# B&R Automation Studio project vibratorControlWithCurrentController (part 13)

#### machine.st - Init, cyclic, exit code
```iecst
PROGRAM _INIT
	cm.setup.name := 'machine';
	cm.setup.parent.name := 'main';

	this.CfgSetIPAddr_0.Option  := cfgOPTION_NON_VOLATILE;
	//this.hmi.setNtpClient := TRUE;

	ST_name(0,ADR(this.configName),0);
	brdkStrCat(ADR(this.configName),ADR(':this.hmi.config'));

	this.hmi.config.dhcpEnabled := TRUE;

	this.TON_updateIp.PT := T#30s;

//	this.forceOutputsFB[0].dpName  := '%QX.IF6.ST6.DigitalOutput01'; //main:this.hw.do_stopButtonIndicator
//	this.forceOutputsFB[1].dpName  := '%QX.IF6.ST6.DigitalOutput02'; //main:this.hw.do_startButtonIndicator
	this.forceOutputsFB[2].dpName  := '%QX.IF6.ST2.DigitalOutput02'; //main:this.hw.do_alarmBeacon
	//this.forceOutputsFB[3].dpName  := '%QX.IF6.ST13.DigitalOutput01'; //feeder:this.hw.do_beltForwards
	//this.forceOutputsFB[4].dpName  := '%QX.IF6.ST13.DigitalOutput02'; //feeder:this.hw.do_beltBackwards
	this.forceOutputsFB[5].dpName  := '%QX.IF6.ST2.DigitalOutput01'; //feeder:this.hw.do_levelSensorInBowlLow
	this.forceOutputsFB[6].dpName  := '%QX.IF6.ST2.DigitalOutput03'; //feeder:this.hw.do_levelSensorInBowlMedium
	this.forceOutputsFB[7].dpName  := '%QX.IF6.ST2.DigitalOutput05'; //feeder:this.hw.do_levelSensorInBowlHigh

	this.forceOutputsFB[8].dpName  := '%QX.IF6.ST7.DigitalOutput01'; //upperFlap:this.hw.do_open
	this.forceOutputsFB[9].dpName  := '%QX.IF6.ST7.DigitalOutput03'; //middleFlap:this.hw.do_open
	this.forceOutputsFB[10].dpName := '%QX.IF6.ST8.DigitalOutput01'; //bottomFlap:this.hw.do_open
	this.forceOutputsFB[11].dpName := '%QX.IF6.ST8.DigitalOutput03'; //bottomFlap:this.hw.do_neighbourOpen
	this.forceOutputsFB[12].dpName := '%QX.IF6.ST7.DigitalOutput04'; //cassette:this.hw.do_dosing
	this.forceOutputsFB[13].dpName := '%QX.IF6.ST8.DigitalOutput05'; //cassette:this.hw.do_cassetteRelease
	this.forceOutputsFB[14].dpName := '%QX.IF6.ST7.DigitalOutput07'; //cassette:this.hw.do_bricksReadyInCassette
	this.forceOutputsFB[15].dpName := '%QX.IF6.ST7.DigitalOutput10'; //external:this.hw.do_itemsDelivered

//	this.forceOutputsFB[16].dpName := '%QX.IF6.ST10.DigitalOutput02'; //feeder:this.hw.do_flapOpen
//	this.forceOutputsFB[17].dpName := '%QX.IF6.ST10.DigitalOutput01'; //feeder:this.hw.do_flapClose
//	this.forceOutputsFB[18].dpName := '%QX.IF6.ST10.DigitalOutput04'; //feeder:this.hw.do_flapClose
//	this.forceOutputsFB[19].dpName := '%QX.IF6.ST10.DigitalOutput03'; //feeder:this.hw.do_flapOpen

	this.forceOutputsFB[20].dpName := '%QX.IF6.ST11.ClearError01'; //belt:this.hw.pwm.clearError
	this.forceOutputsFB[21].dpName := '%QW.IF6.ST11.PulseWidthCurrentPWM01'; //belt:this.hw.pwm.pulseWidth
	hgInfo;
	this.DTGetTime_0.enable := TRUE;

	FOR i:=0 TO MAX_FORCE_OUTPUTS DO
		this.forceOutputsFB[i].setValue := 1;
	END_FOR

	this.hmi.version := hgInfo.version;

	gMainInterface.status.statusIT.Version := CONCAT('CM20 ',this.hmi.version);

END_PROGRAM

PROGRAM _CYCLIC
	IF cm.status.parent.state = STATE_STOPPED THEN
		IF this.forceOutputsFB[16].enable AND this.forceOutputsFB[17].enable THEN	// We can't open all 4 transistors in H-bridge. This will cause a short circuit.
			// if user try to force both - disable both.
			this.forceOutputsFB[16].enable := FALSE;	//feeder flap open
			this.forceOutputsFB[17].enable := FALSE;	//feeder flap close
		END_IF
		this.forceOutputsFB[19].enable := this.forceOutputsFB[16].enable;
		this.forceOutputsFB[18].enable := this.forceOutputsFB[17].enable;

		FOR i:=0 TO MAX_FORCE_OUTPUTS DO
			this.forceOutputsFB[i]();
		END_FOR
	ELSE // Machine not stopped
		FOR i:=0 TO MAX_FORCE_OUTPUTS DO
			this.forceOutputsFB[i].enable := FALSE;
			this.forceOutputsFB[i]();
		END_FOR
	END_IF

	CASE cm.state OF

		0:

			IF NOT gMainInterface.status.simulation  THEN
				IF gFile.status.ready AND (gRecipe.status.saved OR gRecipe.status.loaded) AND (gConfig.status.saved OR gConfig.status.loaded)  THEN
					gConfig.status.loadInitialValue[4] := FALSE;
					this.hmi.config.dhcpEnabled := TRUE; // Machines always have DHCP on servercommunication card.
					cm.state := 10;
				END_IF
			ELSE
				this.hmi.actualLocalIpAddress := this.hmi.config.setLocalIpAddress := '127.0.0.1';
				this.hmi.actualServerIpAddress := this.hmi.config.setServerIpAddress := '127.0.0.2';
			END_IF

		10:
			cm.description := 'get local IP address';

			this.CfgGetIPAddr_0.pDevice := ADR('IF2');
			this.CfgGetIPAddr_0.pIPAddr := ADR(this.hmi.actualLocalIpAddress);
			this.CfgGetIPAddr_0.Len 	:= SIZEOF(this.hmi.actualLocalIpAddress);

			this.CfgGetIPAddr_0(enable := TRUE);

			IF this.CfgGetIPAddr_0.status = ERR_OK THEN
				this.CfgGetIPAddr_0(enable := FALSE);
				this.hmi.actualLocalIpAddress;
				IF brdkStrLen(ADR(this.hmi.config.setLocalIpAddress)) < 7 THEN
					brsstrcpy(ADR(this.hmi.config.setLocalIpAddress),ADR(this.hmi.actualLocalIpAddress));
				END_IF
				cm.state :=  20;
			ELSIF this.CfgGetIPAddr_0.status <> ERR_FUB_BUSY THEN
				recoverState := cm.state;
				cm.state := 9999;
			END_IF

		20:
			cm.description := 'get server IP address';

			this.CfgGetIPAddr_0.pDevice := ADR('SS1.IF1.ETH');
			this.CfgGetIPAddr_0.pIPAddr := ADR(this.hmi.actualServerIpAddress);
			this.CfgGetIPAddr_0.Len 	:= SIZEOF(this.hmi.actualServerIpAddress);

			this.CfgGetIPAddr_0(enable := TRUE);

			IF this.CfgGetIPAddr_0.status = ERR_OK THEN
				this.CfgGetIPAddr_0(enable := FALSE);
				this.hmi.actualServerIpAddress;
				gMachineInterface.parameter.actualServerIP := this.hmi.actualServerIpAddress;
				IF brdkStrLen(ADR(this.hmi.config.setServerIpAddress)) < 7 THEN
					brsstrcpy(ADR(this.hmi.config.setServerIpAddress),ADR(this.hmi.actualServerIpAddress));
				END_IF
				cm.state := 30;
			ELSIF this.CfgGetIPAddr_0.status <> ERR_FUB_BUSY THEN
				recoverState := cm.state;
				cm.state := 9999;
			END_IF

		30:
			cm.description := 'get gateway';

			this.CfgGetDefaultGateway_0.pDevice := ADR('IF2');
			this.CfgGetDefaultGateway_0.pGateway := ADR(this.hmi.actualGatewayAddress);
			this.CfgGetDefaultGateway_0.Len 	:= SIZEOF(this.hmi.actualGatewayAddress);

			this.CfgGetDefaultGateway_0(enable := TRUE);

			IF this.CfgGetDefaultGateway_0.status = ERR_OK THEN
				this.CfgGetDefaultGateway_0(enable := FALSE);
				this.hmi.actualGatewayAddress;
				IF brdkStrLen(ADR(this.hmi.config.setGatewayAddress)) < 7 THEN
					brsstrcpy(ADR(this.hmi.config.setGatewayAddress),ADR(this.hmi.actualGatewayAddress));
				END_IF

				cm.state := 100; // DONT DO NTP RIGHT NOW IN PROD
			ELSIF this.CfgGetDefaultGateway_0.status <> ERR_FUB_BUSY THEN
				recoverState := cm.state;
				cm.state := 9999;
			END_IF

		40:
			cm.description := 'Set time to something wrong to ensure that NTP Client sync with the server';

			this.DTSetTime_0.enable := TRUE;
			this.DTSetTime_0.DT1 := DT#1996-06-23-03:15:00;
			this.DTSetTime_0();

			IF this.DTSetTime_0.status = ERR_OK THEN
				this.DTSetTime_0.enable := FALSE;
				this.DTSetTime_0();

				cm.state := 50;
			ELSIF this.DTSetTime_0.status <> ERR_FUB_BUSY THEN
				recoverState := cm.state;
				cm.state := 9999;
			END_IF

		50:
			cm.description := 'Set ntp server client';

			this.CfgSetNtpClient_0.enable := TRUE;
			this.CfgSetNtpClient_0.start := TRUE;
			this.CfgSetNtpClient_0.pServerAddress1 := ADR(ntpServerIpAddress);
			this.CfgSetNtpClient_0.option := cfgOPTION_VOLATILE;
			this.CfgSetNtpClient_0();

			IF this.CfgSetNtpClient_0.status = ERR_OK THEN
				this.CfgSetNtpClient_0(enable := FALSE);
				cm.state := 100;
			ELSIF this.CfgSetNtpClient_0.status <> ERR_FUB_BUSY THEN
				//error
				recoverState := cm.state;
				cm.state := 9999;
			END_IF

		100:
			cm.description := 'Read IP if it didnt suceed to read doing boot';

			this.TON_updateIp.IN := this.hmi.actualServerIpAddress = '';

			IF this.TON_updateIp.Q THEN			// IF ip or gateway is not set go read untill DHCP has set it.
				this.TON_updateIp.IN := FALSE;
				cm.state := 110; // Go read server IP.
			END_IF
			this.TON_updateIp();

		110:
			cm.description := 'Get ip received from DHCP network and set it on HMI';

			this.CfgGetIPAddr_0.pDevice := ADR('SS1.IF1.ETH');
			this.CfgGetIPAddr_0.pIPAddr := ADR(this.hmi.actualServerIpAddress);
			this.CfgGetIPAddr_0.Len 	:= SIZEOF(this.hmi.actualServerIpAddress);

			this.CfgGetIPAddr_0(enable := TRUE);

			IF this.CfgGetIPAddr_0.status = ERR_OK THEN
				this.CfgGetIPAddr_0(enable := FALSE);
				this.hmi.actualServerIpAddress;
				cm.state := 100;
			ELSIF this.CfgGetIPAddr_0.status <> ERR_FUB_BUSY THEN
				recoverState := cm.state;
				cm.state := 9999;
			END_IF

			// ERROR

		9999:
			cm.description := 'Wait 5min and go to the state where an error happend';

			this.TON_updateIp.IN := TRUE;
			this.TON_updateIp.PT := T#5m;
			this.TON_updateIp();

			IF this.TON_updateIp.Q THEN
				this.TON_updateIp.IN := FALSE;
				this.TON_updateIp();

				this.errorActive := FALSE;
				this.CfgGetIPAddr_0(enable := FALSE);
				this.CfgSetIPAddr_0(enable := FALSE);
				this.CfgSetDefaultGateway_0(enable := FALSE);
				this.CfgSetEthConfigMode_0(enable := FALSE);
				this.CfgSetSubnetMask_0(enable := FALSE);
				this.CfgSetNtpClient_0(enable := FALSE);
				this.CfgGetEthConfigMode_0(enable := FALSE);
				this.DTGetTime_0(enable := FALSE);
				this.DTSetTime_0(enable := FALSE);
				cm.state := recoverState;
			END_IF

	END_CASE

	gMachineInterface.status.imageServerURL := this.hmi.config.imageServerURL;
	legoSTRItemString_Password();

	cm();

	// IF user suceed to login the password wil be saved for 5min and then cleared
	IF EDGEPOS(this.hmi.loginTriggered) THEN
		TON_login.IN := FALSE;
		TON_login();
		TON_login.IN := TRUE;
		TON_login.PT := T#5m;
		this.hmi.loginTriggered := FALSE;
	END_IF

	TON_login();
	IF TON_login.Q THEN
		TON_login.IN := FALSE;
		TON_login();

		legoSTRItemString_Password.value := 30; // 30 means "clear"
		legoSTRItemString_Password.trigger := TRUE;
	END_IF

	IF this.hmi.confirmReboot THEN
		//this.hmi.confirmReboot := FALSE;
		this.warmRestartWU	:= TRUE;
		TON_0.IN := TRUE;
		TON_0.PT := T#1s;
		TON_0();

		// set warmrestart cmd to WU20

		IF TON_0.Q THEN
			TON_0(IN:=FALSE);
			SYSreset(TRUE,1); // 1, warm restart
		END_IF
	END_IF

	IF gConfig.status.doCheckForChanges AND NOT this.oldCheckChangesConfig THEN
		this.MpRecipeRegPar_Config.Enable := TRUE;
		// chek if it has been loade then update old
		IF gMachineInterface.cmd.serialNoDINT > 0 THEN
			this.hmi.config.serialNumber := gMachineInterface.cmd.serialNoDINT;
		END_IF
		gMainInterface.status.statusIT.SerialNo := DINT_TO_UDINT(this.hmi.config.serialNumber); // serialNo status to IT.

		IF gConfig.status.loaded AND NOT this.oldLoaded THEN
			// Initial program load. Set old=new to avoid saving just after a load (makes no sense)
			this.configOld := this.hmi.config;
		END_IF
		this.oldLoaded := gConfig.status.loaded;

		IF NOT gConfig.cmd.save AND gConfig.status.loaded AND (brsmemcmp(ADR(this.hmi.config),ADR(this.configOld),SIZEOF(this.configOld)) <> 0) THEN
			gConfig.cmd.save := TRUE;
			this.configOld := this.hmi.config;
		END_IF

	END_IF
	this.MpRecipeRegPar_Config(MpLink := ADR(mpRecipe), PVName := ADR(this.configName), Category := ADR('config'));
	this.oldCheckChangesConfig := gConfig.status.doCheckForChanges;

	// Get PLC time.
	this.DTGetTime_0();

	// Some services dont work if we are not in prod. This bool can be used for some of these services to "hardcode" their functionality (example LEGO image server -> we will hardcode som image)
	gMachineInterface.status.machineNotInProduction := this.hmi.config.machineNotInProduction;

END_PROGRAM

PROGRAM _EXIT
	this.CfgGetIPAddr_0(enable := FALSE);
	this.CfgSetIPAddr_0(enable := FALSE);
	this.CfgSetDefaultGateway_0(enable := FALSE);
	this.CfgSetEthConfigMode_0(enable := FALSE);
	this.CfgSetSubnetMask_0(enable := FALSE);
	this.CfgSetNtpClient_0(enable := FALSE);
	this.CfgGetEthConfigMode_0(enable := FALSE);
	this.DTGetTime_0(enable := FALSE);
	this.MpRecipeRegPar_Config(Enable:=FALSE);
	this.DTGetTime_0(enable := FALSE);
	this.DTSetTime_0(enable := FALSE);

	FOR i:=0 TO MAX_FORCE_OUTPUTS DO
		this.forceOutputsFB[i](enable := FALSE);
	END_FOR
END_PROGRAM
```

#### local.typ - Local data types
```iecst
TYPE
	config_machine_typ : 	STRUCT
		setLocalIpAddress : STRING[15];
		setGatewayAddress : STRING[15];
		setServerIpAddress : STRING[15];
		ntpServerIpAddress : STRING[40] := 'time.corp.lego.com';
		softwareVersion : STRING[15];
		dhcpEnabled : BOOL;
		serialNumber : DINT;
		selectedLanguage : STRING[40] := 'en'; (*Language selected on the hmi*)
		imageServerURL : STRING[150] := 'https://ip.cz.pac.corp.lego.com/image-service/api/itemimage/getitemimagedata/';
		machineNotInProduction : BOOL;
	END_STRUCT;
	hmi_typ : 	STRUCT
		setLocalIp : BOOL;
		setServerIp : BOOL;
		setGateway : BOOL;
		setNtpClient : BOOL;
		reboot : BOOL;
		reset : BOOL;
		actualLocalIpAddress : STRING[15];
		actualServerIpAddress : STRING[15];
		actualGatewayAddress : STRING[15];
		openRebootDialog : BOOL;
		confirmReboot : BOOL;
		config : config_machine_typ;
		lineID : STRING[80];
		stringNo : USINT;
		showIpSettings : BOOL;
		version : STRING[50];
		loginTriggered : BOOL;
	END_STRUCT;
	local_typ : 	STRUCT
		forceOutputsFB : ARRAY[0..MAX_FORCE_OUTPUTS]OF brdkSimInput;
		CfgGetIPAddr_0 : CfgGetIPAddr;
		CfgSetIPAddr_0 : CfgSetIPAddr;
		CfgSetDefaultGateway_0 : CfgSetDefaultGateway;
		CfgSetNtpClient_0 : CfgSetNtpClient;
		CfgSetSubnetMask_0 : CfgSetSubnetMask;
		hmi : hmi_typ;
		CfgGetDefaultGateway_0 : CfgGetDefaultGateway;
		configOld : config_machine_typ;
		MpRecipeRegPar_Config : MpRecipeRegPar;
		configName : STRING[80];
		setFromConfig : BOOL;
		CfgGetEthConfigMode_0 : CfgGetEthConfigMode;
		CfgSetEthConfigMode_0 : CfgSetEthConfigMode;
		errorActive : BOOL;
		TON_updateIp : TON; (*In DHCP mode we need to read the IP with a certain interval*)
		tmpString : STRING[15];
		dhcpOnBootAndConfigIsStatic : BOOL; (*Special case to handle if dhcp on boot but config is manually set.*)
		DTGetTime_0 : DTGetTime;
		warmRestartWU : BOOL;
		oldCheckChangesConfig : BOOL;
		oldLoaded : BOOL;
		DTSetTime_0 : DTSetTime;
	END_STRUCT;
END_TYPE
```

#### local.var - Local variables
```iecst
VAR
	i : USINT;
END_VAR
VAR CONSTANT
	MAX_EWU_VERSION_BYTES : USINT := 15;
	MAX_FORCE_OUTPUTS : USINT := 21;
END_VAR
VAR
	cm : brdkCM;
	this : local_typ;
	legoSTRItemString_Password : legoSTRItemString;
	TON_0 : TON;
	ntpServerIpAddress : STRING[40] := '192.168.1.199';
	CfgGetNtpcData_0 : CfgGetNtpcData := (len:=14);
	recoverState : UINT;
	TON_login : TON;
END_VAR
```

### build.typ
```iecst
TYPE
 hg_tortoise_typ : STRUCT
  project : STRING[20] := 'CM20';
  asBuildDate : STRING[16] := '27/11/2024';
  asBuildTime : STRING[16] := '15.09.13';
  revision : STRING[20] := '346';
  id : STRING[40] := 'c6a67033e13a+';
  user : STRING[80] := 'brMadsCornelius <mads.andersen@br-automation.com>';
  date : STRING[30] := 'Tue Nov 26 14:00:32 2024 +0100';
  configurationID : STRING[255] := 'CountingMachine';
  version : STRING[255] := '2.1.42';
  summary : STRING[255] := 'Added support for miniHmi';
  tag: STRING[255] := 'RELEASED';
 END_STRUCT;
END_TYPE
```

### build.var
```iecst
VAR
	hgInfo : hg_tortoise_typ;
END_VAR
```

### Program Logical/services/machine/updateCM (IEC)

#### Main.st - Init, cyclic, exit code
```iecst
PROGRAM _INIT
	cm.setup.name := 'updateCM';
	cm.setup.parent.name := 'main';
	//this.hmi.updateTemplates := TRUE; // always update available templates on a boot.
	isBoot := TRUE;
	templateDropdownSelectedIdx;
END_PROGRAM

PROGRAM _CYCLIC

	CASE cm.state OF

		0:
			IF gFile.status.ready THEN
				brdkUpdateManager_0.enable 		:= TRUE;
				cm.state := 5;
			END_IF

		5:
			// Create devLink to FT50

			this.internal.DevLink_0.enable := TRUE;
			this.internal.DevLink_0.pDevice := ADR('PLC');
			this.internal.DevLink_0.pParam := ADR('/SIP=192.168.2.11 /PROTOCOL=ftp /USER=admin /PASSWORD=admin');
			this.internal.DevLink_0();

			IF this.internal.DevLink_0.status = ERR_OK OR this.internal.DevLink_0.status = fiERR_DEVICE_ALREADY_EXIST THEN
				this.internal.handleDevLink := this.internal.DevLink_0.handle;
				this.internal.DevLink_0(enable:=FALSE);
				cm.state := 7;
			ELSIF this.internal.DevLink_0.status <> ERR_FUB_BUSY THEN
				cm.state := 9999;
			END_IF

		7:
			cm.description := 'Delete update folder if it exists';

			this.internal.DirDeleteEx_0.enable := TRUE;
			this.internal.DirDeleteEx_0.pDevice := ADR('PLC');
			this.internal.DirDeleteEx_0.pName := ADR('F:\Default_X20CP04xx');
			this.internal.DirDeleteEx_0();

			IF this.internal.DirDeleteEx_0.status = ERR_OK OR this.internal.DirDeleteEx_0.status = fiERR_DIR_NOT_EXIST THEN
				this.internal.DirDeleteEx_0(enable:=FALSE);
				cm.state := 8;
			ELSIF this.internal.DirDeleteEx_0.status <> ERR_FUB_BUSY THEN
				this.internal.DirDeleteEx_0(enable:=FALSE);
				cm.state := 9999;
			END_IF

		8:
			cm.description := 'Delete update .xml file if it exists';

			this.internal.FileDelete_0.enable := TRUE;
			this.internal.FileDelete_0.pDevice := ADR('PLC');
			this.internal.FileDelete_0.pName := ADR('F:\arnbcfg.xml');
			this.internal.FileDelete_0();

			IF this.internal.FileDelete_0.status = ERR_OK OR this.internal.FileDelete_0.status = fiERR_FILE_NOT_FOUND THEN
				this.internal.FileDelete_0(enable:=FALSE);
				cm.state := 9;
			ELSIF this.internal.FileDelete_0.status <> ERR_FUB_BUSY THEN
				this.internal.FileDelete_0(enable:=FALSE);
				cm.state := 9999;
			END_IF

		9:
			cm.description := 'Disconnect PLC devlink';

			this.internal.DevUnlink_0.enable := TRUE;
			this.internal.DevUnlink_0.handle := this.internal.handleDevLink;
			this.internal.DevUnlink_0();

			IF this.internal.DevUnlink_0.status = ERR_OK THEN
				this.internal.DevUnlink_0(enable:=FALSE);
				cm.state := 10;
			ELSIF this.internal.DevUnlink_0.status <> ERR_FUB_BUSY THEN
				this.internal.DevUnlink_0(enable:=FALSE);
				cm.state := 9999;
			END_IF

		10:
			IF brdkUpdateManager_0.running.version <> '' THEN
				// go check if any update package on update partition
				brdkUpdateManager_0.cmd.checkForUpdate := TRUE;
				cm.state := 20;	// wait state for command.
			END_IF

		20:

			IF brdkUpdateManager_0.status = ERR_OK THEN
				this.status.readyForUpdate := TRUE;
				IF (brdkStrCmp(ADR(brdkUpdateManager_0.update.version),ADR(brdkUpdateManager_0.running.version)) = 0) THEN		// if update version is equal to the running version -> delete package.
					brdkUpdateManager_0.cmd.deleteUpdate := TRUE;
					cm.state := 30;
				ELSE
					// Update package is not equal -> just continue
					cm.state := 100;
				END_IF
			ELSIF brdkUpdateManager_0.status = fiERR_FILE_NOT_FOUND THEN // no file.
				// no file. Error reset and continue to wait state 100.
				brdkUpdateManager_0.cmd.errorReset := TRUE;
				cm.state := 40;
			END_IF

		30:
			IF brdkUpdateManager_0.status = ERR_OK THEN
				// Update package deleted
				this.cmd.writeUpdateInstalledToGateway := TRUE;
				cm.state := 900; // Write to gateway that software just got updated using opcua.
			END_IF

		40:

			IF brdkUpdateManager_0.status = ERR_OK THEN
				// ready
				cm.state := 100;
			END_IF

		100: // Wait state. React on commands

			IF this.cmd.updateCurrentPackage THEN // cmd from gateway to update from software package.
				this.cmd.updateCurrentPackage := FALSE;
				// reset timer
				TON_0.IN := FALSE;
				TON_0.PT := T#4s;
				TON_0();
				cm.state := 110;
			ELSIF this.cmd.checkForUpdate AND gMachineInterface.parameter.actualServerIP <> '' THEN
				TON_0.IN := FALSE;
				TON_0.PT := T#6s;
				TON_0();
				cm.state := 118; // will check for a new update AND .
			ELSIF this.cmd.checkForUpdateInstantly THEN
				this.cmd.checkForUpdateInstantly := FALSE;
				brdkUpdateManager_0.cmd.checkForUpdate := TRUE;
				cm.state := 130;
			ELSIF this.hmi.updateTemplates AND gMachineInterface.parameter.actualServerIP <> '' THEN
				IF isBoot THEN
					isBoot := FALSE;
					cm.state := 900;
				ELSE
					cm.state := 1000;
				END_IF
			ELSIF this.cmd.loadRecipeTemplateFromGateway AND gMachineInterface.parameter.actualServerIP <> '' THEN

				templateDropdownSelectedIdx;
				IF templateDropdownSelectedIdx <= MAX_TEMPLATES_IDX THEN
					startSearchStr := 'text';
					endSearchStr := '"';
					// Take out the fileName from the dataProvider using substring search.
					brdkStrSubStrSearch(ADR(this.hmi.strRecipeTemplate),
					ADR(this.hmi.templateDataProvider[templateDropdownSelectedIdx]),
					ADR(startSearchStr),ADR(endSearchStr),3,TRUE);
					cm.state := 1000;
				ELSE
					// Error will result in out of bounds.
					this.cmd.loadRecipeTemplateFromGateway := FALSE;
				END_IF

			ELSIF this.cmd.saveRecipeTemplateFromGateway AND gMachineInterface.parameter.actualServerIP <> '' THEN
				IF this.hmi.strRecipeTemplateSaveName <> '' THEN
					cm.state := 1000;
				ELSE
					this.cmd.saveRecipeTemplateFromGateway := FALSE;
				END_IF
			ELSIF this.hmi.automatic.save THEN

				IF gMachineInterface.parameter.actualServerIP <> '' THEN
					this.hmi.strRecipeAutoSaveName := UDINT_TO_STRING(gCapconInterface.status.numBricksInPortion);
					IF gVibratorInterface[0].status.machineType = 0 THEN
						tmpString := 'S';
					ELSE // bif cf
						tmpString := 'L';
					END_IF
					brdkStrCat(ADR(this.hmi.strRecipeAutoSaveName),ADR(tmpString));
					tmpString := DINT_TO_STRING(gMainInterface.status.itemTypeId);
					brdkStrCat(ADR(this.hmi.strRecipeAutoSaveName),ADR(tmpString));
					IF gMainInterface.status.itemTypeId <> 0 AND gCapconInterface.status.numBricksInPortion <> 0 THEN
						cm.state := 1000;
					ELSE
						this.hmi.automatic.save := FALSE;
					END_IF
				ELSE
					this.hmi.automatic.save := FALSE;
				END_IF
			ELSIF this.hmi.automatic.overwrite THEN
				this.hmi.automatic.save := TRUE; // Save like normal. We will tell that it is overwrite further down in the opcua client code.
			ELSIF this.hmi.automatic.load THEN
				IF gMachineInterface.parameter.actualServerIP <> '' THEN
					this.hmi.strRecipeAutoLoadName := UDINT_TO_STRING(gCapconInterface.status.numBricksInPortion);
					IF gVibratorInterface[0].status.machineType = 0 THEN
						tmpString := 'S';
					ELSE // bif cf
						tmpString := 'L';
					END_IF
					brdkStrCat(ADR(this.hmi.strRecipeAutoLoadName),ADR(tmpString));
					tmpString := DINT_TO_STRING(gMainInterface.status.itemTypeId);
					brdkStrCat(ADR(this.hmi.strRecipeAutoLoadName),ADR(tmpString));
					IF gCapconInterface.status.numBricksInPortion <> 0 THEN
						cm.state := 1000;
					ELSE
						this.hmi.automatic.load := FALSE;
					END_IF
				ELSE
					this.hmi.automatic.load := FALSE;
				END_IF
			ELSIF this.hmi.updateAllCMs THEN
				IF gMachineInterface.parameter.actualServerIP <> '' THEN
					cm.state := 1000;
				ELSE
					this.hmi.updateAllCMs := FALSE;
				END_IF
			END_IF

		110:
			// Wait 4sec to be 100% sure that gateway has disconnectet OPCUA CLIENT before rebooting the machine.

			TON_0.IN := TRUE;
			TON_0();
			IF TON_0.Q THEN
				TON_0(IN:=FALSE);
				brdkUpdateManager_0.cmd.updateReboot := TRUE; // update from software package on FTP server.
				cm.state := 112;
			END_IF

		112:

			IF brdkUpdateManager_0.status = ERR_OK THEN
				cm.state := 100;
			ELSIF brdkUpdateManager_0.status <> ERR_FUB_BUSY THEN
				// error reset
				brdkUpdateManager_0.cmd.errorReset := TRUE;
				cm.state := 113;
			END_IF

		113:
			// Wait for reset of error
			IF brdkUpdateManager_0.status = ERR_OK THEN
				cm.state := 100;
			END_IF

		(* ------------------------------------------------------------ *)
		(* 				OPCUA. WRITE UPDATE FILESIZE to GATEWAY         *)
		(* ------------------------------------------------------------ *)

		118:
			// wait 6s to make sure FTP is done.
			TON_0.IN := TRUE;
			TON_0();
			IF TON_0.Q THEN
				TON_0(IN:=FALSE);
				brdkUpdateManager_0.cmd.checkForUpdate := TRUE;
				cm.state := 120;
			END_IF

		120:
			IF brdkUpdateManager_0.status = ERR_OK THEN
				IF brdkUpdateManager_0.update.artransferFileSize > 0 THEN
					// Write file size to gateway
					cm.state := 1000;
				ELSE
					// return? No file size (should never happen)
					this.cmd.checkForUpdate := FALSE;
					cm.state := 100;
				END_IF
			ELSIF brdkUpdateManager_0.status = fiERR_FILE_NOT_FOUND THEN // no file.
				// no file. Error reset and continue to wait state 100.
				brdkUpdateManager_0.cmd.errorReset := TRUE;
				cm.state := 121;
			END_IF

		121: // no update file just return

			IF brdkUpdateManager_0.status = ERR_OK THEN
				this.cmd.checkForUpdate := FALSE;
				cm.state := 100;
			END_IF

		130:
			IF brdkUpdateManager_0.status = ERR_OK THEN
				cm.state := 100;
			ELSIF brdkUpdateManager_0.status = fiERR_FILE_NOT_FOUND THEN // no file.
				// no file. Error reset and continue to wait state 100.
				brdkUpdateManager_0.cmd.errorReset := TRUE;
				cm.state := 131;
			END_IF

		131:
			IF brdkUpdateManager_0.status = ERR_OK THEN
				this.cmd.checkForUpdateInstantly := FALSE;
				cm.state := 100;
			END_IF

		(* ------------------------------------------------------------ *)
		(* OPCUA. WRITE TO GATEWAY THAT NEW SOFTWARE HAS BEEN INSTALLED *)
		(* ------------------------------------------------------------ *)

		900:
			// Wait 7s to be sure that machine got IP from DHCP . (if not it's OK, we will call IP FB untill we get one)
			TON_0.IN := cm.state=900;
			TON_0.PT := T#7s;

			IF TON_0.Q AND gMachineInterface.parameter.actualServerIP <> '' THEN
				TON_0.IN := FALSE;
				cm.state := 1000;
			END_IF
			TON_0();

		1000: (* UA_Connect - establish connection to OPC UA Server *)

			this.opcua.UASessionConnectInfo_0.SecurityMsgMode 								:= UASecurityMsgMode_None;
			this.opcua.UASessionConnectInfo_0.SecurityPolicy 								:= UASecurityPolicy_None;
			this.opcua.UASessionConnectInfo_0.TransportProfile 								:= UATP_UATcp;
			this.opcua.UASessionConnectInfo_0.SessionTimeout 								:= T#1m;
			this.opcua.UASessionConnectInfo_0.MonitorConnection 							:= T#10s;
			this.opcua.UASessionConnectInfo_0.UserIdentityToken.UserIdentityTokenType 		:= UAUITT_Anonymous;

			this.opcua.UA_Connect_0.Execute 			:= TRUE;
			tmpString := gMachineInterface.parameter.actualServerIP;
			brdkStrSlice(ADR(tmpString),0,2);
			IF tmpString = '10' THEN
				// test endpoint in odense
				this.opcua.UA_Connect_0.ServerEndpointUrl 	:= 'opc.tcp://10.45.10.199:4840';
			ELSE
				// production endpoint
				this.opcua.UA_Connect_0.ServerEndpointUrl 	:= 'opc.tcp://192.168.1.199:4840';
			END_IF
			this.opcua.UA_Connect_0.SessionConnectInfo 	:= this.opcua.UASessionConnectInfo_0;
			this.opcua.UA_Connect_0.Timeout 				:= T#30s;

			IF this.opcua.UA_Connect_0.Done THEN
				this.opcua.connectionHdl 		:= this.opcua.UA_Connect_0.ConnectionHdl;
				this.opcua.UA_Connect_0.Execute 	:= FALSE;
				cm.state 				:= 1020;
			ELSIF this.opcua.UA_Connect_0.Error THEN
				this.opcua.errorID 				:= this.opcua.UA_Connect_0.ErrorID;
				this.opcua.UA_Connect_0.Execute 	:= FALSE;
				this.opcua.errorRecoverState := cm.state;
				// return to 100 adn reset all cmds - no gateway
				this.cmd.checkForUpdate := FALSE;
				this.cmd.updateCurrentPackage := FALSE;
				this.hmi.updateTemplates := FALSE;
				this.cmd.loadRecipeTemplateFromGateway := FALSE;
				cm.state 				:= 100;
			END_IF

		1020: (* UA_GetNamespaceIndex - read index of required namespace for PVs *)

			this.opcua.UA_GetNamespaceIndex_0.Execute 		:= TRUE;
			this.opcua.UA_GetNamespaceIndex_0.ConnectionHdl	:= this.opcua.connectionHdl;
			this.opcua.UA_GetNamespaceIndex_0.NamespaceUri 	:= 'http://br-automation.com/OpcUa/PLC/PV/';
			this.opcua.UA_GetNamespaceIndex_0.Timeout 		:= this.opcua.UA_Connect_0.Timeout; // same timeout

			IF this.opcua.UA_GetNamespaceIndex_0.Done THEN
				this.opcua.namespaceIndex 					:= this.opcua.UA_GetNamespaceIndex_0.NamespaceIndex;
				this.opcua.UA_GetNamespaceIndex_0.Execute 	:= FALSE;
				cm.state 							:= 1040;
			ELSIF this.opcua.UA_GetNamespaceIndex_0.Error THEN
				this.opcua.errorID								:= this.opcua.UA_GetNamespaceIndex_0.ErrorID;
				this.opcua.UA_GetNamespaceIndex_0.Execute 	:= FALSE;
				this.opcua.errorRecoverState := cm.state;
				cm.state 							:= 3000;
			END_IF

		1040: // wait state

			IF this.cmd.writeUpdateInstalledToGateway THEN

				this.CfgGetIPAddr_0.pDevice := ADR('SS1.IF1.ETH'); //IF2 is local / SS1.IF1.ETH is server commu card.
				this.CfgGetIPAddr_0.pIPAddr := ADR(this.opcua.actualLocalIpAddress);
				this.CfgGetIPAddr_0.Len 	:= SIZEOF(this.opcua.actualLocalIpAddress);

				this.CfgGetIPAddr_0(enable := TRUE);

				IF this.CfgGetIPAddr_0.status = ERR_OK THEN
					this.CfgGetIPAddr_0(enable := FALSE);
					IF this.opcua.actualLocalIpAddress <> '' THEN // String can't be empty
						this.cmd.writeUpdateInstalledToGateway := FALSE;
						cm.state := 1059;
					END_IF
				ELSIF this.CfgGetIPAddr_0.status <> ERR_FUB_BUSY THEN
					this.CfgGetIPAddr_0(enable:=FALSE); // try again -> dhcp get IP from DHCP yet.
				END_IF
			ELSIF this.cmd.checkForUpdate THEN
				cm.state := 1059;
			ELSIF this.cmd.loadRecipeTemplateFromGateway OR this.hmi.automatic.load THEN
				this.CfgGetIPAddr_0.pDevice := ADR('SS1.IF1.ETH'); //IF2 is local / SS1.IF1.ETH is server commu card.
				this.CfgGetIPAddr_0.pIPAddr := ADR(this.opcua.actualLocalIpAddress);
				this.CfgGetIPAddr_0.Len 	:= SIZEOF(this.opcua.actualLocalIpAddress);

				this.CfgGetIPAddr_0(enable := TRUE);

				IF this.CfgGetIPAddr_0.status = ERR_OK THEN
					this.CfgGetIPAddr_0(enable := FALSE);
					IF this.opcua.actualLocalIpAddress <> '' THEN // String can't be empty
						this.cmd.writeUpdateInstalledToGateway := FALSE;
						cm.state := 1057;
					END_IF
				ELSIF this.CfgGetIPAddr_0.status <> ERR_FUB_BUSY THEN
					this.CfgGetIPAddr_0(enable:=FALSE); // try again -> dhcp get IP from DHCP yet.
				END_IF
			ELSIF this.hmi.updateTemplates THEN

				cm.state := 1056;

			ELSIF this.cmd.saveRecipeTemplateFromGateway OR this.hmi.automatic.save THEN
				this.cmd.saveRecipeTemplateFromGateway := FALSE;
				cm.state := 1058;
			ELSIF this.hmi.updateAllCMs THEN
				cm.state := 1061;
			ELSIF this.cmd.disconnect THEN
				this.cmd.disconnect := FALSE;
				cm.state := 1100;
			END_IF

		1056:
			// prepare bulk before write.
			FOR i:=0 TO MAX_UA_VARIABLES DO
				this.opcua.nodeIDWrite[i].NamespaceIndex := this.opcua.namespaceIndex;
				this.opcua.nodeIDWrite[i].IdentifierType := UAIdentifierType_String;
			END_FOR

			// Node1: "write to gateway that we want to update"
			this.opcua.nodeIDWrite[0].Identifier := '::CM20:templateNames';
			this.opcua.variablesWrite[0] := '::updateCM:templateNames';

			this.opcua.UaClt_ReadBulk_0.ConnectionHdl := this.opcua.connectionHdl;
			this.opcua.UaClt_ReadBulk_0.NodeIDCount := 1;
			this.opcua.UaClt_ReadBulk_0.NodeAddInfo := 0;
			this.opcua.UaClt_ReadBulk_0.TimeStamps := 0;
			this.opcua.UaClt_ReadBulk_0.Timeout := this.opcua.UA_Connect_0.Timeout;
			this.opcua.UaClt_ReadBulk_0.Execute := FALSE;

			cm.state := 1070; // go read bulk

		1057:
			// prepare bulk before write.
			FOR i:=0 TO MAX_UA_VARIABLES DO
				this.opcua.nodeIDWrite[i].NamespaceIndex := this.opcua.namespaceIndex;
				this.opcua.nodeIDWrite[i].IdentifierType := UAIdentifierType_String;
			END_FOR
			writeBool := TRUE;
			findIndexInGatewayArray;
			IF this.hmi.automatic.load THEN

				writeUSINT := 5;
				// Node2: String to specify fileName of the recipe template.
				this.hmi.strRecipeAutoLoadName;
				this.opcua.nodeIDWrite[1].Identifier := '::CM20:recipeTemplateNameStr[';
				tmpString := USINT_TO_STRING(this.opcua.indexInGatewayIpArray);
				brdkStrCat(ADR(this.opcua.nodeIDWrite[1].Identifier),ADR(tmpString));
				tmpString := ']';
				brdkStrCat(ADR(this.opcua.nodeIDWrite[1].Identifier),ADR(tmpString));
				this.opcua.variablesWrite[1] := '::updateCM:this.hmi.strRecipeAutoLoadName';
			ELSE
				writeUSINT := UDINT_TO_USINT(this.hmi.selectedTemplateType);
				// Node2: String to specify fileName of the recipe template.
				this.hmi.strRecipeTemplate;
				this.opcua.nodeIDWrite[1].Identifier := '::CM20:recipeTemplateNameStr[';
				tmpString := USINT_TO_STRING(this.opcua.indexInGatewayIpArray);
				brdkStrCat(ADR(this.opcua.nodeIDWrite[1].Identifier),ADR(tmpString));
				tmpString := ']';
				brdkStrCat(ADR(this.opcua.nodeIDWrite[1].Identifier),ADR(tmpString));
				this.opcua.variablesWrite[1] := '::updateCM:this.hmi.strRecipeTemplate';
			END_IF

			// Node1: cmd to load the recipe
			this.opcua.nodeIDWrite[0].Identifier := '::CM20:writeRecipeTemplate[';
			tmpString := USINT_TO_STRING(this.opcua.indexInGatewayIpArray);
			brdkStrCat(ADR(this.opcua.nodeIDWrite[0].Identifier),ADR(tmpString));
			tmpString := ']';
			brdkStrCat(ADR(this.opcua.nodeIDWrite[0].Identifier),ADR(tmpString));
			this.opcua.variablesWrite[0] := '::updateCM:writeBool';

			// Node3: usint to specify which type of recipe we are using (1pcs,2pcs,3pcs,4pcs, BIG CM or automatic)
			this.opcua.nodeIDWrite[2].Identifier := '::recipeLoad:dirRecipeTemplateType';
			this.opcua.variablesWrite[2] := '::updateCM:writeUSINT';

			this.opcua.UaClt_WriteBulk_0.ConnectionHdl := this.opcua.connectionHdl;
			this.opcua.UaClt_WriteBulk_0.NodeIDCount := 3; // write 2 var
			this.opcua.UaClt_WriteBulk_0.NodeAddInfo := 0;
			this.opcua.UaClt_WriteBulk_0.Timeout := this.opcua.UA_Connect_0.Timeout;
			this.opcua.UaClt_WriteBulk_0.Execute := FALSE;

			cm.state := 1060;

		1058:

			// prepare bulk before write.
			FOR i:=0 TO MAX_UA_VARIABLES DO
				this.opcua.nodeIDWrite[i].NamespaceIndex := this.opcua.namespaceIndex;
				this.opcua.nodeIDWrite[i].IdentifierType := UAIdentifierType_String;
			END_FOR

			writeBool := TRUE;
			findIndexInGatewayArray;
			IF this.hmi.automatic.save THEN
				this.hmi.automatic.save := FALSE;
				writeUSINT := 5; // 5 means we should save to automatic folder.
				// Node2: String to specify fileName of the recipe template.
				this.opcua.nodeIDWrite[1].Identifier := '::CM20:recipeTemplateNameStr[';
				tmpString := USINT_TO_STRING(this.opcua.indexInGatewayIpArray);
				brdkStrCat(ADR(this.opcua.nodeIDWrite[1].Identifier),ADR(tmpString));
				tmpString := ']';
				brdkStrCat(ADR(this.opcua.nodeIDWrite[1].Identifier),ADR(tmpString));
				this.opcua.variablesWrite[1] := '::updateCM:this.hmi.strRecipeAutoSaveName';
			ELSE
				writeUSINT := UDINT_TO_USINT(this.hmi.selectedTemplateType);
				// Node2: String to specify fileName of the recipe template.
				this.opcua.nodeIDWrite[1].Identifier := '::CM20:recipeTemplateNameStr[';
				tmpString := USINT_TO_STRING(this.opcua.indexInGatewayIpArray);
				brdkStrCat(ADR(this.opcua.nodeIDWrite[1].Identifier),ADR(tmpString));
				tmpString := ']';
				brdkStrCat(ADR(this.opcua.nodeIDWrite[1].Identifier),ADR(tmpString));
				this.opcua.variablesWrite[1] := '::updateCM:this.hmi.strRecipeTemplateSaveName';
			END_IF

			// Node1: cmd to save the recipe
			this.opcua.nodeIDWrite[0].Identifier := '::CM20:saveRecipeTemplate[';
			tmpString := USINT_TO_STRING(this.opcua.indexInGatewayIpArray);
			brdkStrCat(ADR(this.opcua.nodeIDWrite[0].Identifier),ADR(tmpString));
			tmpString := ']';
			brdkStrCat(ADR(this.opcua.nodeIDWrite[0].Identifier),ADR(tmpString));
			this.opcua.variablesWrite[0] := '::updateCM:writeBool';

			IF NOT this.hmi.automatic.overwrite THEN
				// Node3: usint to specify which type of recipe we are using (1pcs,2pcs,3pcs,4pcs or BIG CM)
				this.opcua.nodeIDWrite[2].Identifier := '::recipeLoad:dirRecipeTemplateType';
				this.opcua.variablesWrite[2] := '::updateCM:writeUSINT';
			ELSE
				// Node3: Tell that it is overwrite (we already know recipeTemplateType - no reason to write again.
				this.hmi.automatic.overwrite := FALSE;
				this.opcua.nodeIDWrite[2].Identifier := '::CM20:overwriteRecipe[';
				tmpString := USINT_TO_STRING(this.opcua.indexInGatewayIpArray);
				brdkStrCat(ADR(this.opcua.nodeIDWrite[2].Identifier),ADR(tmpString));
				tmpString := ']';
				brdkStrCat(ADR(this.opcua.nodeIDWrite[2].Identifier),ADR(tmpString));
				this.opcua.variablesWrite[2] := '::updateCM:writeBool';
			END_IF

			this.opcua.UaClt_WriteBulk_0.ConnectionHdl := this.opcua.connectionHdl;
			this.opcua.UaClt_WriteBulk_0.NodeIDCount := 3; // write 3 var
			this.opcua.UaClt_WriteBulk_0.NodeAddInfo := 0;
			this.opcua.UaClt_WriteBulk_0.Timeout := this.opcua.UA_Connect_0.Timeout;
			this.opcua.UaClt_WriteBulk_0.Execute := FALSE;

			cm.state := 1060; // go write.

		1059:
			writeBool := TRUE;	// Always true.
			// prepare bulk
			this.opcua.nodeIDWrite[0].NamespaceIndex := this.opcua.namespaceIndex;
			this.opcua.nodeIDWrite[0].IdentifierType := UAIdentifierType_String;
			// ::cm20Recipe:newSoftwareInstalled[0]
			IF NOT this.cmd.checkForUpdate THEN
				 // Write that we are updated
				findIndexInGatewayArray;
				this.opcua.nodeIDWrite[0].Identifier := '::CM20:newSoftwareInstalled[';
				tmpString := USINT_TO_STRING(this.opcua.indexInGatewayIpArray);
				brdkStrCat(ADR(this.opcua.nodeIDWrite[0].Identifier),ADR(tmpString));
				tmpString := ']';
				brdkStrCat(ADR(this.opcua.nodeIDWrite[0].Identifier),ADR(tmpString));
				this.opcua.variablesWrite[0] := '::updateCM:writeBool';
			ELSE 	// Write update file size to gateway
				this.opcua.nodeIDWrite[0].Identifier := '::AsGlobalPV:gUpdateFileSize';
				this.opcua.variablesWrite[0] := '::updateCM:brdkUpdateManager_0.update.artransferFileSize';
			END_IF

			this.opcua.UaClt_WriteBulk_0.ConnectionHdl := this.opcua.connectionHdl;
			this.opcua.UaClt_WriteBulk_0.NodeIDCount := 1; // write 1 var
			this.opcua.UaClt_WriteBulk_0.NodeAddInfo := 0;
			this.opcua.UaClt_WriteBulk_0.Timeout := this.opcua.UA_Connect_0.Timeout;
			this.opcua.UaClt_WriteBulk_0.Execute := FALSE;

			cm.state := 1060;

		1061:
			writeBool := TRUE;	// Always true.
			// prepare bulk
			this.opcua.nodeIDWrite[0].NamespaceIndex := this.opcua.namespaceIndex;
			this.opcua.nodeIDWrite[0].IdentifierType := UAIdentifierType_String;

			// Write to gateway that it should update all online machines.
			findIndexInGatewayArray;
			this.opcua.nodeIDWrite[0].Identifier := '::updateSoft:updateAllOnlineCMs';
			this.opcua.variablesWrite[0] := '::updateCM:writeBool';

			this.opcua.UaClt_WriteBulk_0.ConnectionHdl := this.opcua.connectionHdl;
			this.opcua.UaClt_WriteBulk_0.NodeIDCount := 1; // write 1 var
			this.opcua.UaClt_WriteBulk_0.NodeAddInfo := 0;
			this.opcua.UaClt_WriteBulk_0.Timeout := this.opcua.UA_Connect_0.Timeout;
			this.opcua.UaClt_WriteBulk_0.Execute := FALSE;

			cm.state := 1060;

		1060:

			this.opcua.UaClt_WriteBulk_0.Execute 			:= TRUE;
			this.opcua.UaClt_WriteBulk_0.Variables 			:= ADR(this.opcua.variablesWrite);
			this.opcua.UaClt_WriteBulk_0.NodeErrorIDs 		:= ADR(this.opcua.nodeErrorID);
			this.opcua.UaClt_WriteBulk_0.NodeIDs 			:= ADR(this.opcua.nodeIDWrite);
			IF NOT this.opcua.UaClt_WriteBulk_0.Error THEN
				IF this.opcua.UaClt_WriteBulk_0.Done THEN
					this.opcua.UaClt_WriteBulk_0.Execute := FALSE;
					this.cmd.checkForUpdate 				:= FALSE; 	// reset
					this.hmi.updateAllCMs := FALSE;
					IF this.cmd.loadRecipeTemplateFromGateway OR this.hmi.automatic.load THEN
						this.hmi.automatic.load := FALSE;
						this.cmd.loadRecipeTemplateFromGateway 	:= FALSE;	// reset
						gMainInterface.cmd.loadingTemplateRecipe := TRUE;
					END_IF
					this.cmd.disconnect 					:= TRUE;	// Disconnect client. We are done writing.
					cm.state								:= 1040;
				END_IF
			ELSE // error
				this.opcua.errorID := this.opcua.UaClt_WriteBulk_0.ErrorID;
				this.cmd.checkForUpdate 	 	  	 := FALSE; 	// reset
				this.cmd.loadRecipeTemplateFromGateway 	:= FALSE;	// reset
				this.opcua.UaClt_WriteBulk_0.Execute := FALSE;
				this.opcua.errorRecoverState := cm.state;
				cm.state					 := 3000;
			END_IF

		1070: (* Read bulk *)
			this.opcua.UaClt_ReadBulk_0.Execute := TRUE;
			this.opcua.UaClt_ReadBulk_0.NodeIDs := ADR(this.opcua.nodeIDWrite);
			this.opcua.UaClt_ReadBulk_0.Variables := ADR(this.opcua.variablesWrite);
			this.opcua.UaClt_ReadBulk_0.NodeErrorIDs := ADR(this.opcua.nodeErrorID);

			IF NOT this.opcua.UaClt_ReadBulk_0.Error THEN
				IF this.opcua.UaClt_ReadBulk_0.Done THEN
					this.hmi.updateTemplates := FALSE;
					this.opcua.UaClt_ReadBulk_0.Execute := FALSE;
					this.cmd.disconnect := TRUE;

					IF templateNames[this.hmi.selectedTemplateType].strArr[0] <> '' THEN
						// if a template exist.
						count := 0;
						brdkStrMemSet(ADR(this.hmi.templateDataProvider),0,SIZEOF(this.hmi.templateDataProvider));
						FOR k:=0 TO MAX_TEMPLATES_IDX DO
							IF templateNames[this.hmi.selectedTemplateType].strArr[k] <> '' THEN

								this.hmi.templateDataProvider[count] := '{"value":"';
								tmpString := USINT_TO_STRING(count);
								brdkStrCat(ADR(this.hmi.templateDataProvider[count]),ADR(tmpString));
								tmpString := '", "text":"';
								brdkStrCat(ADR(this.hmi.templateDataProvider[count]),ADR(tmpString));
								tmpString := templateNames[this.hmi.selectedTemplateType].strArr[k];
								brdkStrCat(ADR(this.hmi.templateDataProvider[count]),ADR(tmpString));
								tmpString := '"}';
								brdkStrCat(ADR(this.hmi.templateDataProvider[count]),ADR(tmpString));

								count := count + 1;

							ELSE
								EXIT; // exit no more templates on gateway
							END_IF
						END_FOR
					END_IF

					cm.state := 1040;
				END_IF
			ELSE // error
				this.opcua.errorID := this.opcua.UaClt_ReadBulk_0.ErrorID;
				this.hmi.updateTemplates := FALSE;
				this.opcua.UaClt_ReadBulk_0.Execute := FALSE;
				this.opcua.errorRecoverState := cm.state;
				cm.state					 := 3000;
			END_IF

		1100: (* Disconnect opcua client *)
			this.opcua.UA_Disconnect_0.Execute := TRUE;
			this.opcua.UA_Disconnect_0.ConnectionHdl := this.opcua.connectionHdl;
			this.opcua.UA_Disconnect_0.Timeout := this.opcua.UA_Connect_0.Timeout;

			IF this.opcua.UA_Disconnect_0.Done THEN
				this.opcua.connectionHdl := 0;
				this.opcua.UA_Disconnect_0(Execute := FALSE); // This 1 time call it because we will stop calling FBs when state is changed to 100.
				this.cmd.disconnect := FALSE;
				TON_0(IN:=FALSE);
				cm.state := 100; // Go back to 100 and be ready for an update.
			ELSIF this.opcua.UA_Disconnect_0.Error THEN
				this.opcua.errorID := this.opcua.UA_Disconnect_0.ErrorID;
				this.opcua.UA_Disconnect_0.Execute := FALSE;
				this.opcua.errorRecoverState := cm.state;
				cm.state := 3000;
			END_IF

		2000:	// save recipe on gateway

		3000: (* Error *)

			this.opcua.timerConnectionErrorTimeout.IN := FALSE;
			this.opcua.timerConnectionErrorTimeout.PT := T#3s;
			this.opcua.timerConnectionErrorTimeout(); // make sure timer is reset.
			cm.state := 4000;

		4000: (* UA_ConnectionGetStatus - get server status *)

			this.opcua.timerConnectionErrorTimeout.IN := TRUE;

			// Call UA_connectionGetStatus FB every 3sec
			this.opcua.UA_ConnectionGetStatus_0.Execute 			:= this.opcua.timerConnectionErrorTimeout.Q; // If 3s passed start to call FB.
			this.opcua.UA_ConnectionGetStatus_0.ConnectionHdl 		:= this.opcua.connectionHdl;
			this.opcua.UA_ConnectionGetStatus_0.Timeout 			:= this.opcua.UA_Connect_0.Timeout;

			IF this.opcua.UA_ConnectionGetStatus_0.Done THEN

				IF this.opcua.UA_ConnectionGetStatus_0.ConnectionStatus=UACS_Connected AND this.opcua.UA_ConnectionGetStatus_0.ServerState = UASS_Running THEN
					// Return the state it was coming from
					this.opcua.timerConnectionErrorTimeout.IN := FALSE;
					cm.state := this.opcua.errorRecoverState; // return to the state - server is up again.
				END_IF

				// reset FB and timer
				this.opcua.UA_ConnectionGetStatus_0.Execute := FALSE;
				this.opcua.timerConnectionErrorTimeout.IN := FALSE;

			ELSIF this.opcua.UA_ConnectionGetStatus_0.Error THEN
				// 16#A0080000 "PlcOpen_BadConnectionInvalidHdl" -> Happens if losing connection while calling UA_Disconnect. I've chosen to not react on this
				this.opcua.timerConnectionErrorTimeout.IN := FALSE;
				this.opcua.UA_ConnectionGetStatus_0.Execute := FALSE;
			END_IF
			this.opcua.timerConnectionErrorTimeout();

	END_CASE

	IF cm.state > 999 THEN
		this.opcua.UA_Connect_0();
		this.opcua.UA_GetNamespaceIndex_0();
		this.opcua.UaClt_WriteBulk_0();
		this.opcua.UaClt_ReadBulk_0();
		this.opcua.UA_ConnectionGetStatus_0();
		this.opcua.UA_Disconnect_0();

		// Timeout in case we can't write to gateway.
		TON_1.IN := TRUE;
		TON_1.PT := T#2m;
		IF TON_1.Q THEN
			TON_1.IN := FALSE;

			this.opcua.UA_Connect_0(Execute:=FALSE);
			this.opcua.UA_GetNamespaceIndex_0(Execute:=FALSE);
			this.opcua.UaClt_WriteBulk_0(Execute:=FALSE);
			this.opcua.UaClt_ReadBulk_0(Execute:=FALSE);
			this.opcua.UA_ConnectionGetStatus_0(Execute:=FALSE);
			this.opcua.UA_Disconnect_0(Execute:=FALSE);
			this.cmd.writeUpdateInstalledToGateway := FALSE;

			IF this.opcua.connectionHdl <> 0 THEN
				cm.state := 1100;
			ELSE
				// no connectionHdl just return to 0.
				cm.state := 100;
			END_IF
		END_IF

		TON_1();
	ELSE
		TON_1(IN:=FALSE);
	END_IF

	cm();
	IF gFile.status.ready THEN
		brdkUpdateManager_0.pFileDevice := ADR('UPDATE');
		brdkUpdateManager_0();
	END_IF

END_PROGRAM

PROGRAM _EXIT
	brdkUpdateManager_0(enable:=FALSE);
	this.CfgGetIPAddr_0(enable:=FALSE);
END_PROGRAM
```

#### findIndexInGatewayArray.st
```iecst
ACTION findIndexInGatewayArray:
	tmpString := this.opcua.actualLocalIpAddress := gMachineInterface.parameter.actualServerIP;
	brdkStrSlice(ADR(tmpString),10,13);

	CASE STRING_TO_USINT(tmpString) OF

		201: this.opcua.indexInGatewayIpArray := 0;
		202: this.opcua.indexInGatewayIpArray := 1;
		203: this.opcua.indexInGatewayIpArray := 2;
		204: this.opcua.indexInGatewayIpArray := 3;
		205: this.opcua.indexInGatewayIpArray := 4;
		206: this.opcua.indexInGatewayIpArray := 5;
		207: this.opcua.indexInGatewayIpArray := 6;
		208: this.opcua.indexInGatewayIpArray := 7;
		209: this.opcua.indexInGatewayIpArray := 8;
		210: this.opcua.indexInGatewayIpArray := 9;
		211: this.opcua.indexInGatewayIpArray := 10;
		212: this.opcua.indexInGatewayIpArray := 11;
		213: this.opcua.indexInGatewayIpArray := 12;
		214: this.opcua.indexInGatewayIpArray := 13;
		215: this.opcua.indexInGatewayIpArray := 14;
		216: this.opcua.indexInGatewayIpArray := 15;
		217: this.opcua.indexInGatewayIpArray := 16;
		218: this.opcua.indexInGatewayIpArray := 17;
		221: this.opcua.indexInGatewayIpArray := 18;
		222: this.opcua.indexInGatewayIpArray := 19;
		223: this.opcua.indexInGatewayIpArray := 20;
		224: this.opcua.indexInGatewayIpArray := 21;
		225: this.opcua.indexInGatewayIpArray := 22;
		226: this.opcua.indexInGatewayIpArray := 23;
		227: this.opcua.indexInGatewayIpArray := 24;
		228: this.opcua.indexInGatewayIpArray := 25;
		229: this.opcua.indexInGatewayIpArray := 26;
		230: this.opcua.indexInGatewayIpArray := 27;
		231: this.opcua.indexInGatewayIpArray := 28;
		232: this.opcua.indexInGatewayIpArray := 29;
		233: this.opcua.indexInGatewayIpArray := 30;
		234: this.opcua.indexInGatewayIpArray := 31;
		235: this.opcua.indexInGatewayIpArray := 32;
		236: this.opcua.indexInGatewayIpArray := 33;
		237: this.opcua.indexInGatewayIpArray := 34;
		238: this.opcua.indexInGatewayIpArray := 35;

	END_CASE

	IF this.opcua.actualLocalIpAddress='10.45.10.118' OR this.opcua.actualLocalIpAddress='10.45.10.135'  THEN
		this.opcua.indexInGatewayIpArray := 0; // index 0 when testing in Odense
	ELSIF this.opcua.actualLocalIpAddress='10.45.10.119' OR this.opcua.actualLocalIpAddress='10.45.10.141' THEN
		this.opcua.indexInGatewayIpArray := 1; // index 1 when testing in Odense.
	END_IF

END_ACTION
```

#### Types.typ - Local data types
```iecst
TYPE
	local_typ : 	STRUCT
		cmd : local_cmd_typ;
		status : local_status_typ;
		opcua : local_opcua_typ;
		hmi : local_hmi_typ;
		internal : local_internal_typ;
		CfgGetIPAddr_0 : CfgGetIPAddr;
	END_STRUCT;
	local_cmd_typ : 	STRUCT
		updateCurrentPackage : BOOL;
		clearUpdateFolder : BOOL; (*If any update exists delete*)
		writeUpdateInstalledToGateway : BOOL; (*Write bulk to gateway from CM*)
		disconnect : BOOL; (*disconnect client*)
		reset : BOOL; (*Reset client when in error*)
		checkForUpdate : BOOL;
		loadRecipeTemplateFromGateway : BOOL; (*Will load recipe template from gateway.*)
		saveRecipeTemplateFromGateway : BOOL;
		checkForUpdateInstantly : BOOL; (*Will check for update instantly*)
	END_STRUCT;
	local_status_typ : 	STRUCT
		readyForUpdate : BOOL;
		updateFolderCleared : BOOL; (*Folder is cleared*)
	END_STRUCT;
	local_internal_typ : 	STRUCT
		DevLink_0 : DevLink;
		DirDeleteEx_0 : DirDeleteEx;
		FileDelete_0 : FileDelete;
		DevUnlink_0 : DevUnlink;
		handleDevLink : UDINT;
	END_STRUCT;
	local_hmi_typ : 	STRUCT
		strRecipeTemplate : STRING[30];
		strRecipeTemplateSaveName : STRING[30];
		templateDataProvider : ARRAY[0..MAX_TEMPLATES_IDX]OF STRING[100];
		updateTemplates : BOOL;
		selectedTemplateType : templateType_enum; (*0: 1pcs, 1: 2pcs, 2: 3pcs, 3: 4pcs and 4: Big CM*)
		oldSelectedTemplateType : templateType_enum;
		automatic : local_hmi_automatic_typ;
		strRecipeAutoSaveName : STRING[30];
		strRecipeAutoLoadName : STRING[30];
		updateAllCMs : BOOL;
	END_STRUCT;
	local_hmi_automatic_typ : 	STRUCT
		save : BOOL;
		load : BOOL;
		overwrite : BOOL;
		alreadyExists : BOOL;
		confirmLoad : BOOL;
		confirmSave : BOOL;
	END_STRUCT;
	local_opcua_typ : 	STRUCT
		UA_Connect_0 : UA_Connect;
		connectionHdl : DWORD;
		UASessionConnectInfo_0 : UASessionConnectInfo;
		UA_GetNamespaceIndex_0 : UA_GetNamespaceIndex;
		UaClt_WriteBulk_0 : UaClt_WriteBulk;
		UaClt_ReadBulk_0 : UaClt_ReadBulk;
		variablesWrite : ARRAY[0..MAX_UA_VARIABLES]OF STRING[MAX_LENGTH_VARIABLE];
		nodeIDWrite : ARRAY[0..MAX_UA_VARIABLES]OF UANodeID;
		nodeErrorID : ARRAY[0..MAX_UA_VARIABLES]OF DWORD;
		UA_Disconnect_0 : UA_Disconnect;
		actualLocalIpAddress : STRING[15];
		gatewayEndpoint : USINT;
		errorID : DWORD;
		errorRecoverState : UINT;
		namespaceIndex : UINT;
		indexInGatewayIpArray : USINT;
		timerConnectionErrorTimeout : TON;
		UA_ConnectionGetStatus_0 : UA_ConnectionGetStatus;
		connectionStatus : STRING[20];
	END_STRUCT;
	template_recipes_typ : 	STRUCT
		strArr : ARRAY[0..MAX_TEMPLATES_IDX]OF STRING[30];
	END_STRUCT;
	templateType_enum :
		(
		ONE_PIECE,
		TWO_PIECE,
		THREE_PIECE,
		FOUR_PIECE,
		BIG_CM
		);
END_TYPE
```

#### Variables.var - Local variables
```iecst
VAR
	brdkUpdateManager_0 : brdkUpdateManager;
	cm : brdkCM;
	this : local_typ;
	TON_1 : TON;
	TON_0 : TON;
END_VAR
VAR CONSTANT
	MAX_UA_VARIABLES : USINT := 2; (*Up to 3 UA variables can be read/write at once.*)
END_VAR
VAR
	tmpString : STRING[32];
	writeBool : BOOL;
	i : USINT;
	k : USINT;
	templateNames : ARRAY[0..4] OF template_recipes_typ;
END_VAR
VAR CONSTANT
	MAX_TEMPLATES_IDX : USINT := 39;
END_VAR
VAR
	count : USINT;
	isBoot : BOOL;
	templateDropdownSelectedIdx : UINT;
	startSearchStr : STRING[20];
	endSearchStr : STRING[20];
	writeUSINT : USINT;
END_VAR
```

### Program Logical/services/machine/transferConfigToT50 (IEC)

#### Types.typ
```iecst
TYPE
	local_typ : 	STRUCT
		internal : local_internal_typ;
		hmi : local_hmi_typ;
	END_STRUCT;
	local_internal_typ : 	STRUCT
		DevLink_0 : DevLink;
		FileCopy_0 : FileCopy;
		DevUnlink_0 : DevUnlink;
		reset : BOOL;
		cifsParamFT50 : STRING[120];
		handleDevlinkFT50 : UDINT;
		handleDevlinkPLC : UDINT;
		fileNameSrc : STRING[40];
		fileNameDest : STRING[40];
		ftpParamPLC : STRING[120];
		devLinkFT50exists : BOOL;
		devLinkPLCexists : BOOL;
	END_STRUCT;
	local_hmi_typ : 	STRUCT
		status : USINT; (*0: not done, 1: success, 2: error*)
		cantConnectToFT50 : BOOL;
	END_STRUCT;
END_TYPE
```

#### Variables.var
```iecst
VAR
	cm : brdkCM;
	this : local_typ;
END_VAR
```

#### Main.st
```iecst
PROGRAM _INIT
	cm.setup.name := 'transferConfigToT50';
	cm.setup.parent.name := 'main';
	cm.setup.lastActivated := FALSE;
END_PROGRAM

PROGRAM _CYCLIC

	CASE cm.state OF

		0:

			IF gFile.status.ready AND (gConfig.status.saved OR gConfig.status.loaded) THEN
				cm.state := 100;
			END_IF

		100:
			// Wait for cmd

			IF gMachineInterface.cmd.saveConfigToT50 THEN
				// will reset when succeded (otherwise use can enable while again while saving).
				this.internal.cifsParamFT50 := '/SIP=192.168.2.70 /PROTOCOL=cifs /SHARE=usershare /USER=pft50-user /PASSWORD=1234';
				gMachineInterface.status.configSavedToT50 := FALSE;
				this.hmi.status := 0; // not done
				this.hmi.cantConnectToFT50 := FALSE;
				cm.state := 110;
			END_IF

		110:
			// Create devLink to FT50

			this.internal.DevLink_0.enable := TRUE;
			this.internal.DevLink_0.pDevice := ADR('FT50');
			this.internal.DevLink_0.pParam := ADR(this.internal.cifsParamFT50);
			this.internal.DevLink_0();

			IF this.internal.DevLink_0.status = ERR_OK OR this.internal.DevLink_0.status = fiERR_DEVICE_ALREADY_EXIST THEN
				this.internal.handleDevlinkFT50 := this.internal.DevLink_0.handle;
				IF this.internal.DevLink_0.status = fiERR_DEVICE_ALREADY_EXIST THEN
					this.internal.devLinkFT50exists := TRUE;
				ELSE
					this.internal.devLinkFT50exists := FALSE;
				END_IF
				this.internal.DevLink_0(enable:=FALSE);

				this.internal.ftpParamPLC := '/SIP=192.168.2.11 /PROTOCOL=ftp /USER=superuser /PASSWORD=superuser';
				cm.state := 120;
			ELSIF this.internal.DevLink_0.status <> ERR_FUB_BUSY THEN
				cm.state := 9999;
			END_IF

		120:
			// Create DevLink to PLC

			this.internal.DevLink_0.enable := TRUE;
			this.internal.DevLink_0.pDevice := ADR('PLC');
			this.internal.DevLink_0.pParam := ADR(this.internal.ftpParamPLC);
			this.internal.DevLink_0();

			IF this.internal.DevLink_0.status = ERR_OK OR this.internal.DevLink_0.status = fiERR_DEVICE_ALREADY_EXIST THEN
				this.internal.handleDevlinkPLC := this.internal.DevLink_0.handle;
				IF this.internal.DevLink_0.status = fiERR_DEVICE_ALREADY_EXIST THEN
					this.internal.devLinkPLCexists := TRUE;
				ELSE
					this.internal.devLinkPLCexists := FALSE;
				END_IF
				this.internal.DevLink_0(enable:=FALSE);

				this.internal.fileNameSrc := 'F:\config\config.xml';
				this.internal.fileNameDest := 'config.xml';
				cm.state := 130;
			ELSIF this.internal.DevLink_0.status <> ERR_FUB_BUSY THEN
				cm.state := 9999;
			END_IF

		130:
			// FileCopy config from PLC to FT50 panel

			this.internal.FileCopy_0.enable := TRUE;
			this.internal.FileCopy_0.pSrcDev := ADR('PLC');
			this.internal.FileCopy_0.pSrc := ADR(this.internal.fileNameSrc);
			this.internal.FileCopy_0.pDestDev := ADR('FT50');
			this.internal.FileCopy_0.pDest := ADR(this.internal.fileNameDest);
			this.internal.FileCopy_0.option := fiOVERWRITE;
			this.internal.FileCopy_0();

			IF this.internal.FileCopy_0.status = ERR_OK THEN
				this.internal.FileCopy_0(enable:=FALSE);
				cm.state := 140;
			ELSIF this.internal.FileCopy_0.status <> ERR_FUB_BUSY THEN
				cm.state := 9999;
			END_IF

		140:
			// DevUnlink PLC only unlink if the link was created in this task.
			IF NOT this.internal.devLinkPLCexists THEN
				this.internal.DevUnlink_0.enable := TRUE;
				this.internal.DevUnlink_0.handle := this.internal.handleDevlinkPLC;
				this.internal.DevUnlink_0();

				IF this.internal.DevUnlink_0.status = ERR_OK THEN
					this.internal.handleDevlinkPLC := 0;
					this.internal.DevUnlink_0(enable:=FALSE);

					cm.state := 150;
				ELSIF this.internal.DevUnlink_0.status <> ERR_FUB_BUSY THEN
					cm.state := 9999;
				END_IF
			ELSE
				cm.state := 150;
			END_IF
		150:
			// DevUnlink FT50
			IF NOT this.internal.devLinkFT50exists THEN
				this.internal.DevUnlink_0.enable := TRUE;
				this.internal.DevUnlink_0.handle := this.internal.handleDevlinkFT50;
				this.internal.DevUnlink_0();

				IF this.internal.DevUnlink_0.status = ERR_OK THEN
					this.internal.handleDevlinkFT50 := 0;
					this.internal.DevUnlink_0(enable:=FALSE);

					gMachineInterface.cmd.saveConfigToT50 := FALSE;	 // reset cmd before returning to wait state 100
					gMachineInterface.status.configSavedToT50 := TRUE;
					this.hmi.status := 1; // success
					cm.state := 100;
				ELSIF this.internal.DevUnlink_0.status <> ERR_FUB_BUSY THEN
					cm.state := 9999;
				END_IF
			ELSE
				gMachineInterface.cmd.saveConfigToT50 := FALSE;	 // reset cmd before returning to wait state 100
				gMachineInterface.status.configSavedToT50 := TRUE;
				this.hmi.status := 1; // success
				cm.state := 100;
			END_IF

		9999:
			// ERROR
			this.hmi.status := 2;	// error
			this.hmi.cantConnectToFT50 := TRUE;

			gMachineInterface.cmd.saveConfigToT50 := FALSE;

			// Reset everything and go back to state 100
			this.internal.DevLink_0(enable:=FALSE);
			this.internal.DevUnlink_0(enable:=FALSE);
			this.internal.FileCopy_0(enable:=FALSE);
			cm.state := 0;

	END_CASE

	cm();

END_PROGRAM

PROGRAM _EXIT
	this.internal.DevLink_0(enable:=FALSE);
	this.internal.DevUnlink_0(enable:=FALSE);
	this.internal.FileCopy_0(enable:=FALSE);
END_PROGRAM
```

### machineGlobal.var
```iecst
VAR
	gMachineInterface : gMachineInterface_typ;
END_VAR
```

### machineGlobal.typ
```iecst
TYPE
	gMachineInterface_typ : 	STRUCT
		cmd : gMachineInterface_cmd_typ;
		parameter : gMachineInterface_parameter_typ;
		status : gMachineInterface_status_typ;
	END_STRUCT;
	gMachineInterface_cmd_typ : 	STRUCT
		saveConfigToT50 : BOOL;
		requestSaveToT50 : BOOL; (*request will wait untill config is saved and then trigger the "final cmd to saveConfig"*)
		digitalSiloCmdActive : BOOL; (*main -> udpClient (receive heatbeat so we can blink at the same time)*)
		serialNoDINT : DINT; (*FAT settings serial number*)
	END_STRUCT;
	gMachineInterface_status_typ : 	STRUCT
		configSavedToT50 : BOOL;
		imageServerURL : STRING[150];
		heartBeatFromGateway : UDINT;
		machineNotInProduction : BOOL;
	END_STRUCT;
	gMachineInterface_parameter_typ : 	STRUCT
		actualServerIP : STRING[20];
	END_STRUCT;
END_TYPE
```

### Program Logical/services/machine/updateEWU (IEC)

#### updateEWU.st - Init, cyclic, exit code
```iecst
PROGRAM _INIT
	RemoteUpdate_0.IpEndpoint := '192.168.200.21';
	RemoteUpdate_0.CheckVersion := TRUE; // check version 1 time on boot.
END_PROGRAM

PROGRAM _CYCLIC

	RemoteUpdate_0.Enable := gFile.status.ready;
	RemoteUpdate_0();

END_PROGRAM

PROGRAM _EXIT

END_PROGRAM
```

#### local.var - Local variables
```iecst
VAR
	RemoteUpdate_0 : RemoteUpdate;
END_VAR
```

#### LocalFunctions.fun
```iecst
{REDUND_ERROR} FUNCTION_BLOCK RemoteUpdate (* *) (*$GROUP=User,$CAT=User,$GROUPICON=User.png,$CATICON=User.png*)
	VAR_INPUT
		Enable : BOOL;
		IpEndpoint : STRING[32];
		CheckVersion : BOOL; (*Only check version locally and on eWU*)
		PrepareUpdate : {REDUND_UNREPLICABLE} BOOL; (*Check version locally and on eWU and send it afterward with FTP (if different version)*)
		UpdateEWU : BOOL; (*Will tell the eWU to update.*)
	END_VAR
	VAR_OUTPUT
		VersionEWU : STRING[32];
		VersionLocal : STRING[32];
	END_VAR
	VAR_OUTPUT RETAIN
		UpdateReadyOnEWU : BOOL;
	END_VAR
	VAR
		state : USINT;
		EasyUaRead_0 : EasyUaRead;
		EasyUaWrite_0 : EasyUaWrite;
		brdkUpdateCheck_0 : brdkUpdateCheck;
		brdkUpdateDistributeFTP_0 : brdkUpdateDistributeFTP;
		boolTRUE : BOOL := TRUE; (*Used to write a true bool over OPCUA.*)
		TON_0 : TON;
	END_VAR
END_FUNCTION_BLOCK
```

#### RemoteUpdate.st
```iecst
(*  *)
FUNCTION_BLOCK RemoteUpdate

	CASE state OF

		0:
			IF Enable AND IpEndpoint <> '' THEN
				state := 5;
			END_IF

		5:
			IF CheckVersion OR TON_0.Q THEN
				CheckVersion := FALSE;
				TON_0.IN := FALSE;
				VersionEWU := '';
				VersionLocal := '';
				state := 10;
			ELSIF PrepareUpdate THEN
				VersionEWU := '';
				VersionLocal := '';
				state := 10;
			ELSIF UpdateEWU THEN
				UpdateEWU := FALSE;
				UpdateReadyOnEWU := FALSE;
				state := 100;
			END_IF

			// Only using TON after an EWU update.
			TON_0();

		10:
			// Read EWU version using OPCUA
			EasyUaRead_0.Execute := TRUE;
			EasyUaRead_0.ServerEndpointUrl := 'opc.tcp://';
			EasyUaRead_0.ServerEndpointUrl := CONCAT(EasyUaRead_0.ServerEndpointUrl,IpEndpoint);
			EasyUaRead_0.ServerEndpointUrl := CONCAT(EasyUaRead_0.ServerEndpointUrl,':4840');
			EasyUaRead_0.NodeID.NamespaceIndex := 6;
			//EasyUaRead_0.NodeID.Identifier := '::flaps:hmi.version';
			EasyUaRead_0.NodeID.Identifier := '::updateEWU:brdkUpdateManager_0.running.version';
			EasyUaRead_0.NodeID.IdentifierType := UAIdentifierType_String;
			EasyUaRead_0.Variable := '::updateEWU:RemoteUpdate_0.VersionEWU';
			EasyUaRead_0();

			IF EasyUaRead_0.Done THEN
				EasyUaRead_0.Execute := FALSE;
				EasyUaRead_0();
				state := 20;
			ELSIF EasyUaRead_0.Error THEN
				EasyUaRead_0.Execute := FALSE;
				EasyUaRead_0();
				state := 20;
			END_IF

		20:
			brdkUpdateCheck_0.enable := TRUE;
			brdkUpdateCheck_0.pFileDevice := ADR('UPDATEEWU');
			brdkUpdateCheck_0();

			IF brdkUpdateCheck_0.status = ERR_OK THEN
				brdkUpdateCheck_0.enable := FALSE;
				brdkUpdateCheck_0();
				VersionLocal := brdkUpdateCheck_0.version;
				state := SEL(PrepareUpdate,30,40); // if PrepareUpdate go send - otherwise go back.
			ELSIF brdkUpdateCheck_0.status <> ERR_FUB_BUSY THEN
				brdkUpdateCheck_0.enable := FALSE;
				brdkUpdateCheck_0();
				state := SEL(PrepareUpdate,30,40); // if PrepareUpdate go send - otherwise go back.
			END_IF

			// On exit of state
			IF state <> 20 THEN
				PrepareUpdate := FALSE;
			END_IF

		30:
			IF NOT CheckVersion THEN
				state := 5;
			END_IF

		40:
			// Check if versions are different and no version empty.
			IF VersionLocal <> VersionEWU AND VersionLocal <> '' AND VersionEWU <> '' THEN
				UpdateReadyOnEWU := FALSE;
				state := 45;
			ELSE
				state := 5;
			END_IF

		45:
			// Wait for busy before waiting for ERR_OK (because of stupid design where ERR_OK=0 which it is from the start...)
			brdkUpdateDistributeFTP_0.enable := TRUE;
			brdkUpdateDistributeFTP_0.pFileDevice := ADR('UPDATEEWU');
			brdkUpdateDistributeFTP_0.client[0].pIPAddress := ADR(IpEndpoint);
			brdkUpdateDistributeFTP_0.client[0].pUser := ADR('update');
			brdkUpdateDistributeFTP_0.client[0].pPassword := ADR('update');
			brdkUpdateDistributeFTP_0.cmd.distributeUpdate := TRUE;
			brdkUpdateDistributeFTP_0();

			IF brdkUpdateDistributeFTP_0.status = ERR_FUB_BUSY THEN
				state := 50;
			END_IF

		50:
			brdkUpdateDistributeFTP_0.enable := TRUE;
			brdkUpdateDistributeFTP_0.pFileDevice := ADR('UPDATEEWU');
			brdkUpdateDistributeFTP_0.client[0].pIPAddress := ADR(IpEndpoint);
			brdkUpdateDistributeFTP_0.client[0].pUser := ADR('update');
			brdkUpdateDistributeFTP_0.client[0].pPassword := ADR('update');
			brdkUpdateDistributeFTP_0.cmd.distributeUpdate := TRUE;
			brdkUpdateDistributeFTP_0();

			IF brdkUpdateDistributeFTP_0.status = ERR_OK THEN
				brdkUpdateDistributeFTP_0.enable := FALSE;
				brdkUpdateDistributeFTP_0.cmd.distributeUpdate := FALSE;
				brdkUpdateDistributeFTP_0();
				UpdateReadyOnEWU := TRUE;
				state := 60;
			ELSIF brdkUpdateDistributeFTP_0.status <> ERR_FUB_BUSY THEN
				brdkUpdateDistributeFTP_0.enable := FALSE;
				brdkUpdateDistributeFTP_0.cmd.distributeUpdate := FALSE;
				brdkUpdateDistributeFTP_0();
				state := 60;
			END_IF

		60:
			state := 5;

		100:
			// Write to EWU that it should update.
			EasyUaWrite_0.Execute := TRUE;
			EasyUaWrite_0.ServerEndpointUrl := 'opc.tcp://';
			EasyUaWrite_0.ServerEndpointUrl := CONCAT(EasyUaWrite_0.ServerEndpointUrl,IpEndpoint);
			EasyUaWrite_0.ServerEndpointUrl := CONCAT(EasyUaWrite_0.ServerEndpointUrl,':4840');
			EasyUaWrite_0.NodeID.NamespaceIndex := 6;
			EasyUaWrite_0.NodeID.Identifier := '::updateEWU:hmi.update';
			EasyUaWrite_0.NodeID.IdentifierType := UAIdentifierType_String;
			EasyUaWrite_0.Variable := '::updateEWU:RemoteUpdate_0.boolTRUE';
			EasyUaWrite_0();

			IF EasyUaWrite_0.Done THEN
				EasyUaWrite_0.Execute := FALSE;
				EasyUaWrite_0();
				// Check version after 5min to see if it updated.
				TON_0.IN := TRUE;
				TON_0.PT := T#5m;
				state := 5;
			ELSIF EasyUaWrite_0.Error THEN
				EasyUaWrite_0.Execute := FALSE;
				EasyUaWrite_0();
				state := 5;
			END_IF

	END_CASE

END_FUNCTION_BLOCK
```

### Program Logical/services/machine/lampCtrl (IEC)

#### lampCtrl.st - Init, cyclic, exit code
```iecst
PROGRAM _INIT

	RTInfo_0(enable := TRUE);

	lampIOLink.setOwnColor := TRUE;
	lampIOLink.setBrightness := TRUE;
END_PROGRAM

PROGRAM _CYCLIC

	// call rt info to get cycle time of current task
	IF RTInfo_0.status <> ERR_OK THEN
		RTInfo_0();
	END_IF

	// change the flash for every flash time elapsed
	flash.elapsedTime := flash.elapsedTime + RTInfo_0.cycle_time;
	IF NOT flash.on THEN
		IF flash.elapsedTime >= (config.flash.offTime*1000) THEN
			flash.elapsedTime 	:= 0;
			flash.on 			:= TRUE;
		END_IF
	ELSE
		IF flash.elapsedTime >= (config.flash.onTime*1000) THEN
			flash.elapsedTime 	:= 0;
			flash.on 			:= FALSE;
		END_IF
	END_IF

	// change the blink for every flash time elapsed
	blink.elapsedTime := blink.elapsedTime + RTInfo_0.cycle_time;
	IF NOT blink.on THEN
		IF blink.elapsedTime >= (config.blink.offTime*1000) THEN
			blink.elapsedTime 	:= 0;
			blink.on 			:= TRUE;
		END_IF
	ELSE
		IF blink.elapsedTime >= (config.blink.onTime*1000) THEN
			blink.elapsedTime 	:= 0;
			blink.on 			:= FALSE;
		END_IF
	END_IF

	(*****************************

	IO HANDLING

	*****************************)

	lamp.timeoutActive := FALSE;		// tmp set it to false
	// based on the flash or the color sets the right output to the lamp io
	CASE lamp.flash OF

		FLASH_PERMANENT:
			lamp.io.output := DINT_TO_USINT(lamp.color);

		FLASH_FLASH:
			IF NOT flash.on THEN
				lamp.io.output := DINT_TO_USINT(COLOR_OFF);
			ELSE
				lamp.io.output := DINT_TO_USINT(lamp.color);
			END_IF

		FLASH_BLINK:
			IF NOT blink.on THEN
				lamp.io.output := DINT_TO_USINT(COLOR_OFF);
			ELSE
				lamp.io.output := DINT_TO_USINT(lamp.color);
			END_IF

	END_CASE

	IF lamp.color <> COLOR_OFF THEN
		lamp.timeoutActive := TRUE;
	END_IF

	// store the actual color and flash in the status structure which is remanent
	statusString.lamp.color 	:= lamp.color;
	statusString.lamp.flash		:= lamp.flash;

	(*****************************

	IO-LINK PARAMETERS

	*****************************)

	IF gConfig.status.loaded THEN

		CASE lampIOLink.state OF

				0:	// waiting for command
					lampIOLink.elapsedTime := lampIOLink.elapsedTime + RTInfo_0.cycle_time;
					IF lampIOLink.setBrightness THEN
						IF config.brightness.green <> 0 OR config.brightness.red <> 0 OR config.brightness.blue <> 0 THEN
							lampIOLink.setBrightness 				:= FALSE;
							lampIOLink.ioLinkWrite_0(enable := FALSE);
							lampIOLink.data[0] 					:= LIMIT(0,UINT_TO_USINT((USINT_TO_UINT(config.brightness.red)*127)/100),127);	// 100% = 127
							lampIOLink.data[1] 					:= LIMIT(0,UINT_TO_USINT((USINT_TO_UINT(config.brightness.green)*127)/100),127);	// 100% = 127
							lampIOLink.data[2] 					:= LIMIT(0,UINT_TO_USINT((USINT_TO_UINT(config.brightness.blue)*127)/100),127);	// 100% = 127
							lampIOLink.ioLinkWrite_0.index 		:= 16#51;			// set brightness
							lampIOLink.ioLinkWrite_0.subIndex		:= 1;
							lampIOLink.ioLinkWrite_0.datatype		:= ioLinkTYPE_USINT;
							lampIOLink.ioLinkWrite_0.pData		:= ADR(lampIOLink.data[0]);
							lampIOLink.ioLinkWrite_0.dataLen		:= SIZEOF(lampIOLink.data[0]);
							lampIOLink.ioLinkWrite_0.pDeviceName 	:= ADR(lampIOLink.deviceName);
							lampIOLink.node						:= 2;
							lampIOLink.subIndex					:= 1;
							lampIOLink.stringNo					:= 0; // 0 = G01, 1 = G02

						//							brdkStrCpy(ADR(lampIOLink.deviceName),ADR('IF6.ST'));
						//							brdkStrAppendUdintToA(lampIOLink.node,ADR(lampIOLink.deviceName),BRDK_STR_CONVERT_DECIMAL,-1);
						//							brdkStrCat(ADR(lampIOLink.deviceName),ADR('.IF'));
						//							brdkStrAppendUdintToA(cIdx+1,ADR(lampIOLink.deviceName),BRDK_STR_CONVERT_DECIMAL,-1);
							lampIOLink.deviceName := 'IF6.ST1.IF2';

							lampIOLink.ioLinkWrite_0.enable		:= TRUE;
							lampIOLink.state						:= 10;
						END_IF
					ELSIF lampIOLink.setOwnColor THEN
						IF config.ownColor.green <> 0 OR config.ownColor.red <> 0 OR config.ownColor.blue <> 0 THEN
							lampIOLink.setOwnColor 				:= FALSE;
							lampIOLink.ioLinkWrite_0(enable := FALSE);
							lampIOLink.data[0]					:= config.ownColor.red;
							lampIOLink.data[1]					:= config.ownColor.green;
							lampIOLink.data[2]					:= config.ownColor.blue;
							lampIOLink.ioLinkWrite_0(enable := FALSE);
							lampIOLink.ioLinkWrite_0.index 		:= 16#FC;				// set own color
							lampIOLink.ioLinkWrite_0.subIndex		:= 1;
							lampIOLink.ioLinkWrite_0.datatype		:= ioLinkTYPE_USINT;
							lampIOLink.ioLinkWrite_0.pData		:= ADR(lampIOLink.data[0]);
							lampIOLink.ioLinkWrite_0.dataLen		:= SIZEOF(lampIOLink.data[0]);
							lampIOLink.ioLinkWrite_0.pDeviceName 	:= ADR(lampIOLink.deviceName);
							lampIOLink.node						:= 2;
							lampIOLink.subIndex					:= 1;
							lampIOLink.stringNo					:= 0; // 0 = G01, 1 = G02
//							brdkStrCpy(ADR(lampIOLink.deviceName),ADR('IF6.ST'));
//							brdkStrAppendUdintToA(lampIOLink.node,ADR(lampIOLink.deviceName),BRDK_STR_CONVERT_DECIMAL,-1);
//							brdkStrCat(ADR(lampIOLink.deviceName),ADR('.IF'));
//							brdkStrAppendUdintToA(cIdx+1,ADR(lampIOLink.deviceName),BRDK_STR_CONVERT_DECIMAL,-1);
							lampIOLink.deviceName := 'IF6.ST1.IF2';
							lampIOLink.ioLinkWrite_0.enable		:= TRUE;
							lampIOLink.state						:= 10;
						END_IF
					ELSIF lampIOLink.elapsedTime >= 60000000 THEN	// read temperature only every minute
						lampIOLink.ioLinkRead_0(enable := FALSE);
						lampIOLink.ioLinkRead_0.index 		:= 16#59;				// read temperature
						lampIOLink.ioLinkRead_0.subIndex		:= 1;
						lampIOLink.ioLinkRead_0.datatype		:= ioLinkTYPE_SINT;
						lampIOLink.ioLinkRead_0.pData			:= ADR(lampIOLink.temperature);
						lampIOLink.ioLinkRead_0.dataLen		:= SIZEOF(lampIOLink.temperature);
						lampIOLink.ioLinkRead_0.pDeviceName 	:= ADR(lampIOLink.deviceName);
						lampIOLink.node						:= 2;
						lampIOLink.stringNo					:= 0; // 0 = G01, 1 = G02
//						brdkStrCpy(ADR(lampIOLink.deviceName),ADR('IF6.ST'));
//						brdkStrAppendUdintToA(lampIOLink.node,ADR(lampIOLink.deviceName),BRDK_STR_CONVERT_DECIMAL,-1);
//						brdkStrCat(ADR(lampIOLink.deviceName),ADR('.IF'));
//						brdkStrAppendUdintToA(cIdx+1,ADR(lampIOLink.deviceName),BRDK_STR_CONVERT_DECIMAL,-1);
						lampIOLink.deviceName := 'IF6.ST1.IF2';
						lampIOLink.ioLinkRead_0.enable		:= TRUE;
						lampIOLink.temperature				:= 0;
						lampIOLink.state						:= 20;
					END_IF

				10: // wait for ioLinkWrite_0 status ok
					lampIOLink.ioLinkWrite_0();

//					IF lampIOLink[2].node = 1 THEN
//						lampIOLink[2].node := lampIOLink[2].node;
//					END_IF

					CASE lampIOLink.ioLinkWrite_0.status OF

						ERR_OK,ioLinkERR_COMMUNICATION_DEVICE,ioLinkERR_INVALID_MASTER,ioLinkERR_DEVICE_DRIVER:
							lampIOLink.ioLinkWrite_0(enable := FALSE);
							lampIOLink.ioLinkWrite_0.enable		:= TRUE;
							lampIOLink.elapsedTime 	:= 0; // ADDED
							lampIOLink.state := 0; // ADDED
						(*
							lampIOLink.subIndex := lampIOLink.subIndex + 1;
							IF lampIOLink.subIndex > 3 THEN
								lampIOLink.subIndex 	:= 1;
								lampIOLink.node		:= lampIOLink.node + 1;

								CASE lampIOLink.stringNo OF

									0: // G01 - IF6.ST2 -> IF6.ST7
										IF NOT di_G04_10_08Present THEN // SSPP line or DSPP line
											IF lampIOLink.node > 7 THEN
												IF NOT di_G02Present THEN	// SSPP line - only one string
													lampIOLink.state := 0;
												ELSE
													lampIOLink.node						:= 1;
													lampIOLink.subIndex					:= 1;
													lampIOLink.stringNo					:= 1; // 0 = G01, 1 = G02
													brdkStrCpy(ADR(lampIOLink.deviceName),ADR('SS1.IF1.ST'));
												END_IF
											ELSE
												brdkStrCpy(ADR(lampIOLink.deviceName),ADR('IF6.ST'));
											END_IF
										ELSE	// PP99 line
											IF lampIOLink.node > 9 THEN
												lampIOLink.node						:= 1;
												lampIOLink.subIndex					:= 1;
												lampIOLink.stringNo					:= 1; // 0 = G01, 1 = G02
												brdkStrCpy(ADR(lampIOLink.deviceName),ADR('SS1.IF1.ST'));
											ELSE
												brdkStrCpy(ADR(lampIOLink.deviceName),ADR('IF6.ST'));
											END_IF
										END_IF

									1: // G02 - SS1.IF1.ST1 -> SS1.IF1.ST6
										IF NOT di_G04_10_08Present THEN // DSPP line
											IF lampIOLink.node > 6 THEN
												lampIOLink.elapsedTime 	:= 0;
												lampIOLink.state 			:= 0;
											ELSE
												brdkStrCpy(ADR(lampIOLink.deviceName),ADR('SS1.IF1.ST'));
											END_IF
										ELSE	// PP99 line
											IF lampIOLink.node > 8 THEN
												lampIOLink.elapsedTime 	:= 0;
												lampIOLink.state 			:= 0;
											ELSE
												brdkStrCpy(ADR(lampIOLink.deviceName),ADR('SS1.IF1.ST'));
											END_IF
										END_IF

								END_CASE

								IF lampIOLink.state > 0 THEN
									brdkStrAppendUdintToA(lampIOLink.node,ADR(lampIOLink.deviceName),BRDK_STR_CONVERT_DECIMAL,-1);
									brdkStrCat(ADR(lampIOLink.deviceName),ADR('.IF'));
									brdkStrAppendUdintToA(cIdx+1,ADR(lampIOLink.deviceName),BRDK_STR_CONVERT_DECIMAL,-1);
								END_IF

							END_IF
							*)
							lampIOLink.ioLinkWrite_0.subIndex 	:= lampIOLink.subIndex;
							lampIOLink.ioLinkWrite_0.pData		:= ADR(lampIOLink.data[lampIOLink.ioLinkWrite_0.subIndex-1]);

					END_CASE

				20:	// wait for ioLinkRead_0 status ok
					lampIOLink.ioLinkRead_0();
					CASE lampIOLink.ioLinkRead_0.status OF

						ERR_OK,ioLinkERR_COMMUNICATION_DEVICE,ioLinkERR_INVALID_MASTER,ioLinkERR_DEVICE_DRIVER:
							lampIOLink.ioLinkRead_0(enable := FALSE);
							lampIOLink.ioLinkRead_0.enable		:= TRUE;
							lampIOLink.elapsedTime 	:= 0;
							lampIOLink.state 			:= 0;

//							setTemperature; // call action
//							lampIOLink.temperature := 0;
//							lampIOLink.node		:= lampIOLink.node + 1;
//
//							CASE lampIOLink.stringNo OF
//
//								0: // G01 - IF6.ST2 -> IF6.ST7
//									IF NOT di_G04_10_08Present THEN // SSPP line or DSPP line
//										IF lampIOLink.node > 7 THEN
//											IF NOT di_G02Present THEN	// SSPP line - only one string
//												lampIOLink.elapsedTime 	:= 0;
//												lampIOLink.state 			:= 0;
//											ELSE
//												lampIOLink.node						:= 1;
//												lampIOLink.stringNo					:= 1; // 0 = G01, 1 = G02
//												brdkStrCpy(ADR(lampIOLink.deviceName),ADR('SS1.IF1.ST'));
//											END_IF
//										ELSE
//											brdkStrCpy(ADR(lampIOLink.deviceName),ADR('IF6.ST'));
//										END_IF
//									ELSE	// PP99 line
//										IF lampIOLink.node > 9 THEN
//											lampIOLink.node						:= 1;
//											lampIOLink.stringNo					:= 1; // 0 = G01, 1 = G02
//											brdkStrCpy(ADR(lampIOLink.deviceName),ADR('SS1.IF1.ST'));
//										ELSE
//											brdkStrCpy(ADR(lampIOLink.deviceName),ADR('IF6.ST'));
//										END_IF
//									END_IF
//
//								1: // G02 - SS1.IF1.ST1 -> SS1.IF1.ST6
//									IF NOT di_G04_10_08Present THEN // DSPP line
//										IF lampIOLink.node > 6 THEN
//											lampIOLink.elapsedTime 	:= 0;
//											lampIOLink.state 			:= 0;
//										ELSE
//											brdkStrCpy(ADR(lampIOLink.deviceName),ADR('SS1.IF1.ST'));
//										END_IF
//									ELSE // PP99 line
//										IF lampIOLink.node > 8 THEN
//											lampIOLink.elapsedTime 	:= 0;
//											lampIOLink.state 			:= 0;
//										ELSE
//											brdkStrCpy(ADR(lampIOLink.deviceName),ADR('SS1.IF1.ST'));
//										END_IF
//									END_IF
//
//							END_CASE
//
//							IF lampIOLink.state > 0 THEN
//								brdkStrAppendUdintToA(lampIOLink.node,ADR(lampIOLink.deviceName),BRDK_STR_CONVERT_DECIMAL,-1);
//								brdkStrCat(ADR(lampIOLink.deviceName),ADR('.IF'));
//								brdkStrAppendUdintToA(cIdx+1,ADR(lampIOLink.deviceName),BRDK_STR_CONVERT_DECIMAL,-1);
//							END_IF
//
					END_CASE

			END_CASE

	END_IF

//	// copy status vlaue to tmp variable for multiple outputs
//	tmpLamp1_1 := plcString[1].lamp[1].io.status;
//	tmpLamp1_4 := plcString[1].lamp[4].io.status;
//
//	(*****************************
//
//	STATUS
//
//	*****************************)
//	// brightness
//	Lamp.Status.Configuration.Brightness.Blue 	:= config.brightness.blue;
//	Lamp.Status.Configuration.Brightness.Green 	:= config.brightness.green;
//	Lamp.Status.Configuration.Brightness.Red 	:= config.brightness.red;
//
//	// own color
//	Lamp.Status.Configuration.OwnColor.Blue 	:= config.ownColor.blue;
//	Lamp.Status.Configuration.OwnColor.Green 	:= config.ownColor.green;
//	Lamp.Status.Configuration.OwnColor.Red 		:= config.ownColor.red;
//
//	// health check
//	Lamp.Status.Configuration.HealthCheck.ColorTimeout := config.healthCheck.timeout;
//	FOR sIdx := 0 TO 6 DO
//		Lamp.Status.Configuration.HealthCheck.ColorSequence[sIdx].Color := config.healthCheck.colorSequence[sIdx];
//	END_FOR
//
//	// test position
//	Lamp.Status.Configuration.TestPosition.Color := config.testPosition.color;
//	Lamp.Status.Configuration.TestPosition.Timeout := config.testPosition.timeout;
//
//	// flashing
//	Lamp.Status.Configuration.Flashing.Permanent.Timeout.Time 	:= config.permanent.timeout;
//	Lamp.Status.Configuration.Flashing.Flash.Timeout.Time		:= config.flash.timeout;
//	Lamp.Status.Configuration.Flashing.Flash.TimeOn.Time		:= config.flash.onTime;
//	Lamp.Status.Configuration.Flashing.Flash.TimeOff.Time		:= config.flash.offTime;
//	Lamp.Status.Configuration.Flashing.Blink.Repeat				:= config.blink.repeat;
//	Lamp.Status.Configuration.Flashing.Blink.TimeOn.Time		:= config.blink.onTime;
//	Lamp.Status.Configuration.Flashing.Blink.TimeOff.Time		:= config.blink.offTime;
//
//	gStatus;
//
//	MpRecipeRegPar_Config.MpLink 	:= ADR(gRecipeXmlConfig);
//	MpRecipeRegPar_Config.Enable 	:= TRUE;
//	MpRecipeRegPar_Config.PVName 	:= ADR('::lampCtrl:config');
//	MpRecipeRegPar_Config.Category 	:= ADR('config');
//	MpRecipeRegPar_Config();

END_PROGRAM

PROGRAM _EXIT

END_PROGRAM
```

#### local.typ - Local data types
```iecst
(*Lamp*)

TYPE
	plc_lamp_typ : 	STRUCT
		color : lamp_color_typ; (*Activate color*)
		flash : lamp_flash_typ; (*Activate flash*)
		temperature : SINT; (*Read temperature*)
		io : plc_lamp_io_typ; (*I/O structure*)
		timeoutActive : BOOL;
		timeoutElapsedTime : UDINT;
	END_STRUCT;
	lamp_color_typ :
		(
		COLOR_OFF := 0, (*NO COLOR*)
		COLOR_GREEN := 1, (*GREEN*)
		COLOR_RED := 2, (*RED*)
		COLOR_YELLOW := 3, (*YELLOW*)
		COLOR_BLUE := 4, (*BLUE*)
		COLOR_ORANGE := 5, (*ORANGE*)
		COLOR_OWN := 6, (*OWN*)
		COLOR_WHITE := 7 (*WHITE*)
		) := COLOR_OFF;
	lamp_flash_typ :
		(
		FLASH_PERMANENT := 0,
		FLASH_FLASH := 1,
		FLASH_BLINK := 2
		) := FLASH_PERMANENT;
	plc_lamp_io_typ : 	STRUCT
		output : USINT; (*Variable mapped to X67DS438A module*)
		status : USINT; (*Variable mapped to X67DS438A module*)
	END_STRUCT;
	status_string_typ : 	STRUCT
		lamp : status_lamp_typ;
	END_STRUCT;
	status_lamp_typ : 	STRUCT
		color : lamp_color_typ; (*Activate color*)
		flash : lamp_flash_typ; (*Activate flash*)
		repeat : UDINT;
		timeout : UDINT;
	END_STRUCT;
	flash_typ : 	STRUCT
		elapsedTime : UDINT;
		on : BOOL;
	END_STRUCT;
END_TYPE

(*config*)

TYPE
	config_typ : 	STRUCT
		brightness : config_color_typ;
		ownColor : config_color_typ;
		healthCheck : config_healthcheck_typ;
		permanent : config_permanent_typ;
		testPosition : config_test_position_typ;
		flash : config_flash_typ;
		blink : config_blink_typ;
	END_STRUCT;
	config_lamp_typ : 	STRUCT
		subStringNo : UDINT;
	END_STRUCT;
	config_permanent_typ : 	STRUCT
		timeout : UDINT := 120000; (*2min*)
	END_STRUCT;
	config_flash_typ : 	STRUCT
		timeout : UDINT := 120000; (*2min*)
		onTime : UDINT := 1000; (*1s*)
		offTime : UDINT := 1000; (*1s*)
	END_STRUCT;
	config_blink_typ : 	STRUCT
		onTime : UDINT := 1000; (*1s*)
		offTime : UDINT := 1000; (*1s*)
		repeat : UDINT;
	END_STRUCT;
	config_healthcheck_typ : 	STRUCT
		colorSequence : ARRAY[0..6]OF lamp_color_typ := [COLOR_GREEN,COLOR_BLUE,COLOR_ORANGE,COLOR_RED,COLOR_WHITE,2(COLOR_OFF)];
		timeout : UDINT := 10000; (*10s*)
	END_STRUCT;
	config_color_typ : 	STRUCT
		blue : USINT := 100;
		green : USINT := 100;
		red : USINT := 100;
	END_STRUCT;
	config_test_position_typ : 	STRUCT
		color : lamp_color_typ := COLOR_GREEN; (*Activate color*)
		timeout : UDINT := 2000; (*2s*)
	END_STRUCT;
END_TYPE

(*IO-LINK communication*)

TYPE
	lamp_iolink_typ : 	STRUCT
		state : DINT;
		ioLinkWrite_0 : ioLinkWrite;
		ioLinkRead_0 : ioLinkRead;
		setBrightness : BOOL;
		setOwnColor : BOOL;
		data : ARRAY[0..2]OF USINT;
		deviceName : STRING[80];
		node : USINT;
		subIndex : USINT;
		temperature : SINT;
		stringNo : USINT;
		elapsedTime : UDINT;
	END_STRUCT;
END_TYPE
```

#### local.var - Local variables
```iecst
VAR
	config : config_typ;
	lamp : plc_lamp_typ;
END_VAR
VAR RETAIN
	statusString : status_string_typ;
END_VAR
VAR
	blink : flash_typ;
	flash : flash_typ;
	lampIOLink : lamp_iolink_typ;
	RTInfo_0 : RTInfo;
END_VAR
```

### Program Logical/services/machine/udpClient (IEC)

#### Main.st - Init, cyclic, exit code
```iecst
PROGRAM _INIT

END_PROGRAM

PROGRAM _CYCLIC

	(*
	-----------------------------------------------------------------------------------------------------------------------------------------------------------
	---------------------------------------- UDP client implementation to synchronize blinking of digital silo cards. ----------------------------------------
	-----------------------------------------------------------------------------------------------------------------------------------------------------------
	The server will broadcast an incrementing UDINT to the subnet (192.168.1.xxx) with a time interval specified in "lampCtrl".
	The client (CM20) will then receive this UDINT making it possible to blink simultaneously.
	-----------------------------------------------------------------------------------------------------------------------------------------------------------
	-----------------------------------------------------------------------------------------------------------------------------------------------------------
	-----------------------------------------------------------------------------------------------------------------------------------------------------------
	*)

	CASE Client.sStep OF

		0:
			IF gMachineInterface.cmd.digitalSiloCmdActive THEN
				Client.sStep := 5;
			END_IF

		5:	(* Open UDP Port *)
			Client.UdpOpen_0.enable := TRUE;
			Client.UdpOpen_0.pIfAddr := 0;	(* Listen on all TCP/IP Interfaces*)
			Client.UdpOpen_0.port := 12058;	(* Port to listen*)
			Client.UdpOpen_0.options := udpOPT_BROADCAST;
			Client.UdpOpen_0();

			IF Client.UdpOpen_0.status = 0 THEN  (* UdpOpen successful*)
				Client.sStep := 10;
			ELSIF Client.UdpOpen_0.status = ERR_FUB_BUSY THEN  (* UdpOpen not finished -> redo *)
				(* Busy *)
			ELSE  (* Goto Error Step *)
				Client.sStep := 222;
			END_IF

		10:	(* Receive Data from the Server *)
			Client.UdpRecv_0.enable := TRUE;
			Client.UdpRecv_0.ident := Client.UdpOpen_0.ident;  (* Connection Ident from AsUDP.UDP_Open *)
			Client.UdpRecv_0.pData	:= ADR(receive_data);  (* Where to store the incoming data *)
			Client.UdpRecv_0.datamax := SIZEOF(receive_data);  (* Lenght of data buffer *)
			Client.UdpRecv_0.pIpAddr := ADR(Client.server_address);
			Client.UdpRecv_0.flags := 0;
			Client.UdpRecv_0();  (* Call the Function*)

			IF Client.UdpRecv_0.status = 0 THEN  (* Data was received successfully -> Send next packet *)

				// Check that package is coming from the correct IP
				IF gMachineInterface.cmd.digitalSiloCmdActive THEN
					IF Client.server_address='192.168.1.199' OR Client.server_address='192.168.30.207' THEN // Gateway in prod or test IP in Odense
						gMachineInterface.status.heartBeatFromGateway := receive_data;
					END_IF
				ELSE
					// Digital silo not active - close the port.
					Client.sStep := 20;
				END_IF

			ELSIF Client.UdpRecv_0.status = udpERR_NO_DATA THEN  (* No data received - wait *)
				(* No Data received *)
			ELSIF Client.UdpRecv_0.status = ERR_FUB_BUSY THEN  (* UdpRecv not finished -> redo *)
				(* Busy *)
			ELSE  (* Goto Error Step *)
				Client.sStep := 222;
			END_IF

		20: (* Close connection *)
			Client.UdpClose_0.enable := TRUE;
			Client.UdpClose_0.ident := Client.UdpOpen_0.ident;  (* Connection Ident from AsUDP.UDP_Open *)
			Client.UdpClose_0();

			IF Client.UdpClose_0.status = 0 THEN  (* Close successful -> Reopen the interface *)
				Client.sStep := 0;
			ELSIF Client.UdpClose_0.status = ERR_FUB_BUSY THEN  (* UdpClose not finished -> redo *)
				(* Busy *)
			ELSE  (* Goto Error Step *)
				Client.sStep := 222;
			END_IF

		222: (* Here some error Handling has to be implemented *)

	END_CASE

END_PROGRAM

PROGRAM _EXIT
	(* Insert code here *)

END_PROGRAM
```

#### usdSync.typ - Local data types
```iecst
TYPE
	Client_typ : 	STRUCT  (*UDP Client Variables*)
		sStep : UINT; (*UDP Client Step Variable*)
		server_address : STRING[20]; (*Address of the Server*)
		server_portnumber : UINT; (*Portnumber of the Server*)
		no_data_received_count : UINT; (*Counts up if no data are received*)
		UdpOpen_0 : UdpOpen; (*AsUDP.UdpOpen FUB*)
		UdpConnect_0 : UdpConnect; (*AsUDP.UdpConnect FUB*)
		UdpSend_0 : UdpSend; (*AsUDP.UdpSend FUB*)
		UdpRecv_0 : UdpRecv; (*AsUDP.UdpRecv FUB*)
		UdpDisconnect_0 : UdpDisconnect; (*AsUDP.UdpDisconnect FUB*)
		UdpClose_0 : UdpClose; (*AsUDP.UdpClose FUB*)
	END_STRUCT;
END_TYPE
```

#### udpSync.var - Local variables
```iecst
VAR
	Client : Client_typ := (0); (*Data for Client Task*)
	receive_data : UDINT;
END_VAR
```

### Package Logical/services/language - project language definition

- project.language - project langugae definition file (not shown)

### Package Logical/services/alarm - This module is used to handle all machine alarms.

### alarmGlobal.typ - Global data types
```iecst
TYPE
	gAlarm_status_typ : 	STRUCT  (*Status of the alarm module.*)
		ready : BOOL := FALSE; (*Alarm module is ready to use.*)
	END_STRUCT;
	gAlarm_typ : 	STRUCT  (*Global alarm interface.*)
		status : gAlarm_status_typ; (*Status of the alarm module.*)
		cmd : gAlarm_cmd_typ;
	END_STRUCT;
	gAlarm_struct_typ : 	STRUCT
		name : STRING[255];
		active : BOOL;
		oldActive : BOOL;
		instanceID : UDINT;
	END_STRUCT;
	gAlarm_cmd_typ : 	STRUCT  (*Commands for alarm module*)
		acknowledgeAll : BOOL; (*Acknowledge all alarms*)
		acknowledge : BOOL; (*Acknowledge selected alarm on HMI*)
		exportLogToCsv : BOOL;
	END_STRUCT;
END_TYPE
```

### alarmGlobal.var - Global variables
```iecst
VAR
	gAlarm : gAlarm_typ; (*Global alarm module interface.*)
END_VAR
```

### Program Logical/services/alarm/alarm (IEC, version 1.00.0) - alarm system

#### alarm.st - Init, cyclic, exit code
```iecst
PROGRAM _INIT

	cm.setup.name			:= 'alarm';
	cm.setup.parent.name 	:= 'main';
	gAlarm.status.ready		:= FALSE;

END_PROGRAM

PROGRAM _CYCLIC

	IF MpAlarmXCore_0.Error THEN
		cm.state := 9999;
	END_IF

	CASE cm.state OF

		0:
			cm.description 	:= 'wait for MpAlarmXCore and MpAlarmXListUI_0 to be active';

			IF MpAlarmXCore_0.Active AND gFile.status.ready THEN
				MpAlarmXHistory_0.Enable := TRUE;
				cm.state 	:= 100;
			END_IF

		100:
			cm.description 		:= 'alarm system ready';

			gAlarm.status.ready	:= TRUE;

			TON_0.IN := TRUE;;
			TON_0.PT := T#30m;
			TON_0();

			IF gAlarm.cmd.acknowledge THEN
				AlarmXListUIConnectType.Acknowledge := TRUE;
				gAlarm.cmd.acknowledge := FALSE;
			ELSIF gAlarm.cmd.acknowledgeAll THEN
				AlarmXListUIConnectType.AcknowledgeAll := TRUE;
				gAlarm.cmd.acknowledgeAll := FALSE;
			ELSIF gAlarm.cmd.exportLogToCsv OR TON_0.Q THEN
				TON_0.IN := gAlarm.cmd.exportLogToCsv := FALSE;
				TON_0();
				logAlarmsError := FALSE;
				cm.state := 200;
			END_IF

		200:
			cm.description := '';

			DevLink_0.enable := TRUE;
			DevLink_0.pDevice := ADR('PLC');
			DevLink_0.pParam := ADR('/SIP=192.168.2.11 /PROTOCOL=ftp /USER=admin /PASSWORD=admin');
			DevLink_0();

			IF DevLink_0.status = ERR_OK OR DevLink_0.status = fiERR_DEVICE_ALREADY_EXIST THEN
				DevLink_0(enable:=FALSE);
				cm.state := 210;
			ELSIF DevLink_0.status <> ERR_FUB_BUSY THEN
				DevLink_0(enable:=FALSE);
				logAlarmsError := TRUE;
				cm.state := 100;
			END_IF

		210:
			DirDeleteEx_0.enable := TRUE;
			DirDeleteEx_0.pDevice := ADR('PLC');
			DirDeleteEx_0.pName := ADR('F:\alarm');
			DirDeleteEx_0();

			IF DirDeleteEx_0.status = ERR_OK OR DirDeleteEx_0.status = fiERR_DIR_NOT_EXIST THEN
				DirDeleteEx_0(enable:=FALSE);
				cm.state := 220;
			ELSIF DirDeleteEx_0.status <> ERR_FUB_BUSY THEN
				DirDeleteEx_0(enable:=FALSE);
				logAlarmsError := TRUE;
				cm.state := 100;
			END_IF

		220:
			DirCreate_0.enable := TRUE;
			DirCreate_0.pDevice := ADR('PLC');
			DirCreate_0.pName := ADR('F:\alarm');
			DirCreate_0();

			IF DirCreate_0.status = ERR_OK THEN
				DirCreate_0(enable:=FALSE);
				MpAlarmXHistory_0.Export := TRUE;
				cm.state := 230;
			ELSIF DirCreate_0.status <> ERR_FUB_BUSY THEN
				DirCreate_0(enable:=FALSE);
				logAlarmsError := TRUE;
				cm.state := 100;
			END_IF

		230:
			IF MpAlarmXHistory_0.CommandDone THEN
				MpAlarmXHistory_0.Export := FALSE;
				cm.state := 100;
			ELSIF MpAlarmXHistory_0.Error THEN
				MpAlarmXHistory_0.Enable := FALSE;
				MpAlarmXHistory_0.Export := FALSE;
				logAlarmsError := TRUE;
				cm.state := 100;
			END_IF

		9999:
			cm.description 	:= 'wait for error reset';

			MpAlarmXCore_0.ErrorReset := TRUE;

			IF NOT MpAlarmXCore_0.Error THEN
				MpAlarmXCore_0.ErrorReset := FALSE;
				cm.state 	:= 0;
			END_IF

	END_CASE

	cm();

//	MpAlarmXListUI_0.MpLink := ADR(mpAlarmXCore);
//	MpAlarmXListUI_0.Enable := TRUE;
//	MpAlarmXListUI_0.UIConnect := ADR(AlarmXListUIConnectType);
//	MpAlarmXListUI_0.UISetup := AlarmXListUISetupType;
//	MpAlarmXListUI_0();

	MpAlarmXCore_0.Enable := TRUE;
	MpAlarmXCore_0.MpLink := ADR(mpAlarmXCore);
	MpAlarmXCore_0();

	MpAlarmXHistory_0.MpLink := ADR(mpAlarmXHistory);
	MpAlarmXHistory_0.DeviceName := ADR('ALARM');
	MpAlarmXHistory_0();

END_PROGRAM

PROGRAM _EXIT
	MpAlarmXListUI_0(Enable:=FALSE);
	MpAlarmXCore_0(Enable := FALSE);
	MpAlarmXHistory_0(Enable:=FALSE);
END_PROGRAM
```

#### local.var - Local variables
```iecst
VAR
	cm : brdkCM; (*Control module.*)
	MpAlarmXCore_0 : MpAlarmXCore; (*MpAlarmXCore function block.*)
	MpAlarmXHistory_0 : MpAlarmXHistory;
	AlarmXListUIConnectType : MpAlarmXListUIConnectType;
	MpAlarmXListUI_0 : MpAlarmXListUI;
	TON_0 : TON;
	DevLink_0 : DevLink;
	DirDeleteEx_0 : DirDeleteEx;
	logAlarmsError : BOOL;
	DirCreate_0 : DirCreate;
END_VAR
```

### Package Logical/services/file - This module is used to handle all file devices.

### fileGlobal.typ - Global data types
```iecst
TYPE
	gFile_typ : 	STRUCT  (*Global file type.*)
		cmd : gFile_cmd_typ; (*File command type.*)
		status : gFile_status_typ; (*File status type.*)
	END_STRUCT;
	gFile_status_typ : 	STRUCT  (*File status type.*)
		ready : BOOL; (*File devices are ready to use.*)
	END_STRUCT;
	gFile_cmd_typ : 	STRUCT  (*File command type.*)
		update : BOOL; (*Update file devices command.*)
	END_STRUCT;
END_TYPE
```

### fileGlobal.var - Global variables
```iecst
VAR
	gFile : gFile_typ; (*Global file interface.*)
END_VAR
```

### Program Logical/services/file/file (IEC, version 1.00.0) - file device management task

#### file.st - Init, cyclic, exit code
```iecst
PROGRAM _INIT

	cm.setup.name			:= 'file';
	cm.setup.parent.name 	:= 'main';
	gFile.status.ready 		:= FALSE;
	gFile.cmd.update 		:= FALSE;

	// add file device used for the data logging
	brdkFileDeviceHandler_0.setup.fileDevices[0].name := 'CONFIG';
	brdkFileDeviceHandler_0.setup.fileDevices[0].path := 'config';
	brdkFileDeviceHandler_0.setup.fileDevices[1].name := 'RECIPES';
	brdkFileDeviceHandler_0.setup.fileDevices[1].path := 'recipes';
	brdkFileDeviceHandler_0.setup.fileDevices[2].name := 'DATA';
	brdkFileDeviceHandler_0.setup.fileDevices[2].path := 'data';
	brdkFileDeviceHandler_0.setup.fileDevices[3].name := 'IMAGES';
	brdkFileDeviceHandler_0.setup.fileDevices[3].path := 'images';
	brdkFileDeviceHandler_0.setup.fileDevices[4].name := 'ALARM';
	brdkFileDeviceHandler_0.setup.fileDevices[4].path := 'alarm';
	brdkFileDeviceHandler_0.setup.fileDevices[5].name := 'REPORT';
	brdkFileDeviceHandler_0.setup.fileDevices[5].path := 'report';
	brdkFileDeviceHandler_0.setup.fileDevices[6].name := 'UPDATE';
	brdkFileDeviceHandler_0.setup.fileDevices[6].path := 'update';
	brdkFileDeviceHandler_0.setup.fileDevices[7].name := 'UPDATEEWU';
	brdkFileDeviceHandler_0.setup.fileDevices[7].path := 'updateewu';
	brdkFileDeviceHandler_0.setup.fileDevices[8].name := 'RESULT';
	brdkFileDeviceHandler_0.setup.fileDevices[8].path := 'result';

	// file devices are automatically created on a USB drive whenever it is inserted.
	brdkFileDeviceHandler_0.setup.usbOverrule := FALSE;

	//brdkFileDeviceHandler_0.simulation.pcUSBDrive		:= E_DRIVE;
	IF gMainInterface.status.simulation THEN
		brdkFileDeviceHandler_0.setup.plcDrive := C_DRIVE;
	ELSE
		brdkFileDeviceHandler_0.setup.plcDrive := F_DRIVE;
	END_IF

END_PROGRAM

PROGRAM _CYCLIC

	CASE cm.state OF

		0:
			cm.description := 'wait for brdkFileDeviceHandler to be done detecting file devices';

			brdkFileDeviceHandler_0.enable 	:= TRUE;
			gFile.status.ready := FALSE;
			IF brdkFileDeviceHandler_0.ready THEN
				cm.state := 100;
			ELSIF brdkFileDeviceHandler_0.status <> 0 THEN
				cm.state := 9999;
			END_IF

		100:
			cm.description := 'wait for commands';

			gFile.status.ready := TRUE;

			IF gFile.cmd.update THEN
				gFile.status.ready := FALSE;
				gFile.cmd.update := FALSE;
				brdkFileDeviceHandler_0.enable := FALSE;
				cm.state := 110;
			END_IF

		110:
			cm.description := 'wait for brdkFileDeviceHandler to be disabled';

			IF NOT brdkFileDeviceHandler_0.ready THEN
				cm.state := 0;
			END_IF

		9999:
			cm.description := 'wait for error reset';

			IF brdkFileDeviceHandler_0.status = 0 THEN
				cm.state := 0;
			END_IF

	END_CASE

	cm();
	brdkFileDeviceHandler_0();

END_PROGRAM

PROGRAM _EXIT

	brdkFileDeviceHandler_0(enable := FALSE);

END_PROGRAM
```

#### local.var - Local variables
```iecst
VAR
	cm : brdkCM; (*Control module.*)
	brdkFileDeviceHandler_0 : brdkFileDeviceHandler; (*brdkFileDeviceHandler function block.*)
END_VAR
```

### Package Logical/services/recipe - This module is used to handle all machine recipes.

### recipeGlobal.typ - Global data types
```iecst
TYPE
	gRecipe_typ : 	STRUCT  (*Global recipe type.*)
		cmd : gRecipe_cmd_typ; (*Command type.*)
		status : gRecipe_status_typ; (*Status type.*)
	END_STRUCT;
	gRecipe_cmd_typ : 	STRUCT  (*Global command type.*)
		load : BOOL; (*Load command.*)
		saveCurrent : BOOL; (*Save current recipe to file of RECIPES partition*)
		save : BOOL; (*Save command.*)
		loadCurrent : BOOL; (*Load current recipe to file of RECIPES partition*)
		brickID : STRING[80]; (*BrickID for the recipe to load.*)
	END_STRUCT;
	gRecipe_status_typ : 	STRUCT  (*Global status type.*)
		saved : BOOL; (*Recipe saved.*)
		loaded : BOOL; (*Recipe loaded.*)
		doCheckForChanges : BOOL;
		newRecipeLoaded : BOOL;
	END_STRUCT;
END_TYPE
```

### recipeGlobal.var - Global variables
```iecst
VAR
	gRecipe : gRecipe_typ; (*Global recipe interface.*)
END_VAR
```

### Program Logical/services/recipe/recipe (IEC, version 1.00.0) - recipe management
